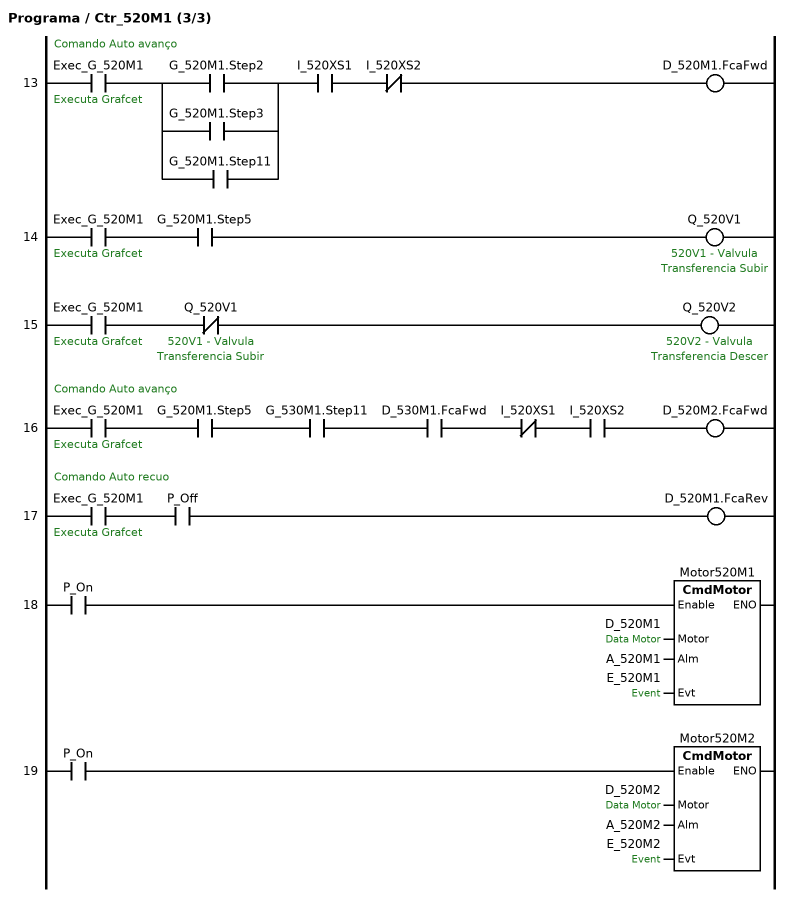
(* [picture p120: Programa / Ctr_520M1, rungs 13-19] *)
(* Rung 13: Comando Auto avanço *)
D_520M1.FcaFwd := Exec_G_520M1 AND (G_520M1.Step2 OR G_520M1.Step3 OR G_520M1.Step11) AND I_520XS1 AND NOT I_520XS2;
(* Rung 14 *)
Q_520V1 := Exec_G_520M1 AND G_520M1.Step5;
(* Rung 15 *)
Q_520V2 := Exec_G_520M1 AND NOT Q_520V1;
(* Rung 16: Comando Auto avanço *)
D_520M2.FcaFwd := Exec_G_520M1 AND G_520M1.Step5 AND G_530M1.Step11 AND D_530M1.FcaFwd AND NOT I_520XS1 AND I_520XS2;
(* Rung 17: Comando Auto recuo *)
D_520M1.FcaRev := Exec_G_520M1 AND P_Off;
(* Rung 18 *)
Motor520M1(Enable := P_On, Motor := D_520M1, Alm := A_520M1, Evt := E_520M1);
(* Rung 19 *)
Motor520M2(Enable := P_On, Motor := D_520M2, Alm := A_520M2, Evt := E_520M2);

(* Section Ctr_530M1: ladder, written here as Structured Text *)

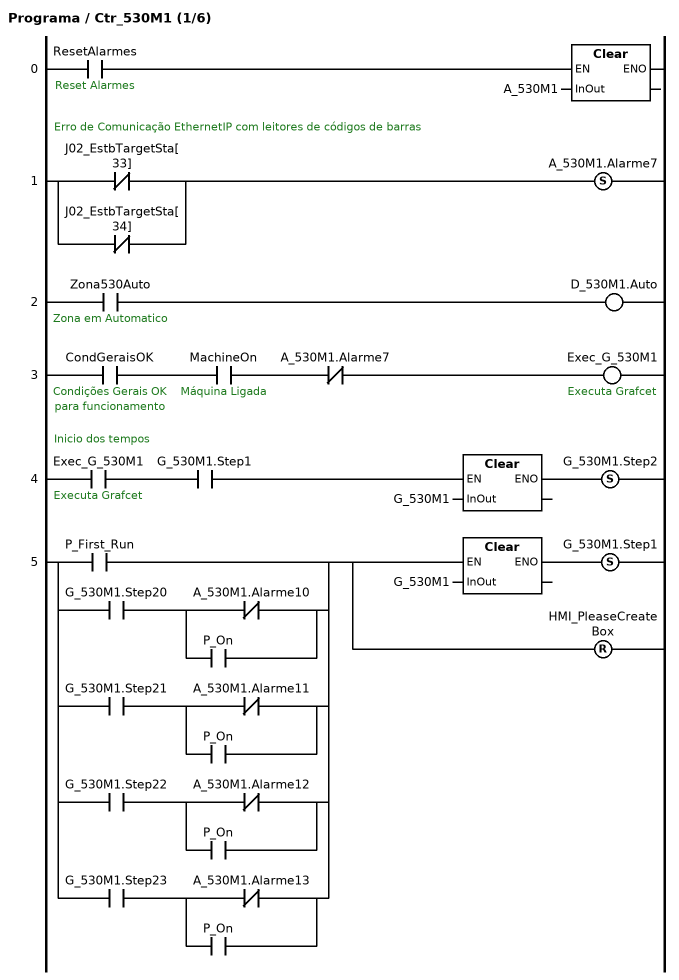
(* Rung 0 *)
IF ResetAlarmes THEN Clear(InOut := A_530M1); END_IF;
(* Rung 1: Erro de Comunicação EthernetIP com leitores de códigos de barras *)
IF NOT J02_EstbTargetSta[33] OR NOT J02_EstbTargetSta[34] THEN A_530M1.Alarme7 := TRUE; END_IF;
(* Rung 2 *)
D_530M1.Auto := Zona530Auto;
(* Rung 3 *)
Exec_G_530M1 := CondGeraisOK AND MachineOn AND NOT A_530M1.Alarme7;
(* Rung 4: Inicio dos tempos *)
_p223 := Exec_G_530M1 AND G_530M1.Step1;
IF _p223 THEN
    Clear(InOut := G_530M1);
    G_530M1.Step2 := TRUE;
END_IF;
(* Rung 5 *)
_p224 := P_First_Run OR (G_530M1.Step20 AND (NOT A_530M1.Alarme10 OR P_On)) OR (G_530M1.Step21 AND (NOT A_530M1.Alarme11 OR P_On)) OR (G_530M1.Step22 AND (NOT A_530M1.Alarme12 OR P_On)) OR (G_530M1.Step23 AND (NOT A_530M1.Alarme13 OR P_On));
IF _p224 THEN
    Clear(InOut := G_530M1);
    G_530M1.Step1 := TRUE;
    HMI_PleaseCreateBox := FALSE;
END_IF;

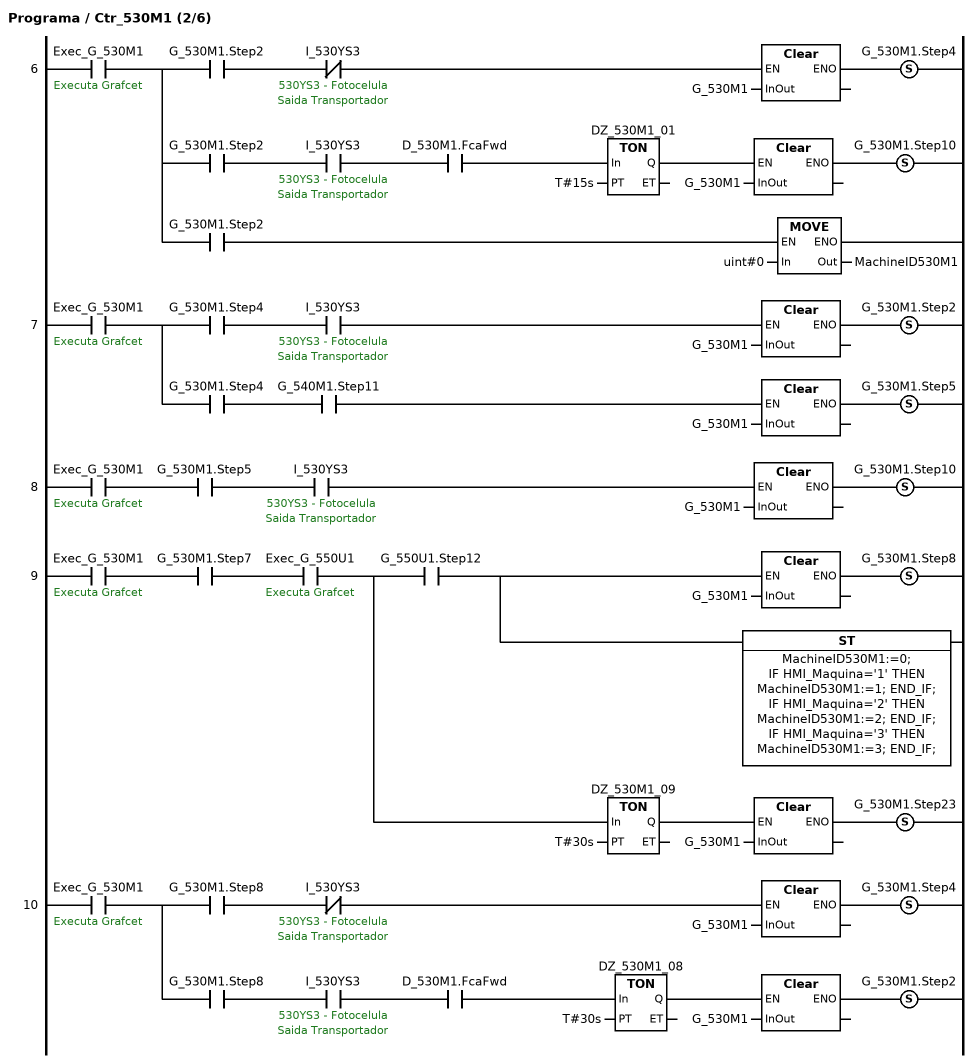
(* Rung 6 *)
_p225 := Exec_G_530M1 AND G_530M1.Step2 AND NOT I_530YS3;
IF _p225 THEN
    Clear(InOut := G_530M1);
    G_530M1.Step4 := TRUE;
END_IF;
DZ_530M1_01(In := Exec_G_530M1 AND G_530M1.Step2 AND I_530YS3 AND D_530M1.FcaFwd, PT := T#15s);
IF DZ_530M1_01.Q THEN
    Clear(InOut := G_530M1);
    G_530M1.Step10 := TRUE;
END_IF;
IF Exec_G_530M1 AND G_530M1.Step2 THEN MachineID530M1 := uint#0; END_IF;
(* Rung 7 *)
_p226 := Exec_G_530M1 AND G_530M1.Step4 AND I_530YS3;
IF _p226 THEN
    Clear(InOut := G_530M1);
    G_530M1.Step2 := TRUE;
END_IF;
_p227 := Exec_G_530M1 AND G_530M1.Step4 AND G_540M1.Step11;
IF _p227 THEN
    Clear(InOut := G_530M1);
    G_530M1.Step5 := TRUE;
END_IF;
(* Rung 8 *)
_p228 := Exec_G_530M1 AND G_530M1.Step5 AND I_530YS3;
IF _p228 THEN
    Clear(InOut := G_530M1);
    G_530M1.Step10 := TRUE;
END_IF;
(* Rung 9 *)
_p229 := Exec_G_530M1 AND G_530M1.Step7 AND Exec_G_550U1 AND G_550U1.Step12;
_p230 := Exec_G_530M1 AND G_530M1.Step7 AND Exec_G_550U1;
IF _p229 THEN
    Clear(InOut := G_530M1);
    G_530M1.Step8 := TRUE;
END_IF;
IF _p229 THEN
    MachineID530M1:=0;
    IF HMI_Maquina='1' THEN MachineID530M1:=1; END_IF;
    IF HMI_Maquina='2' THEN MachineID530M1:=2; END_IF;
    IF HMI_Maquina='3' THEN MachineID530M1:=3; END_IF;
END_IF;
DZ_530M1_09(In := _p230, PT := T#30s);
IF DZ_530M1_09.Q THEN
    Clear(InOut := G_530M1);
    G_530M1.Step23 := TRUE;
END_IF;
(* Rung 10 *)
_p231 := Exec_G_530M1 AND G_530M1.Step8 AND NOT I_530YS3;
IF _p231 THEN
    Clear(InOut := G_530M1);
    G_530M1.Step4 := TRUE;
END_IF;
DZ_530M1_08(In := Exec_G_530M1 AND G_530M1.Step8 AND I_530YS3 AND D_530M1.FcaFwd, PT := T#30s);
IF DZ_530M1_08.Q THEN
    Clear(InOut := G_530M1);
    G_530M1.Step2 := TRUE;
END_IF;

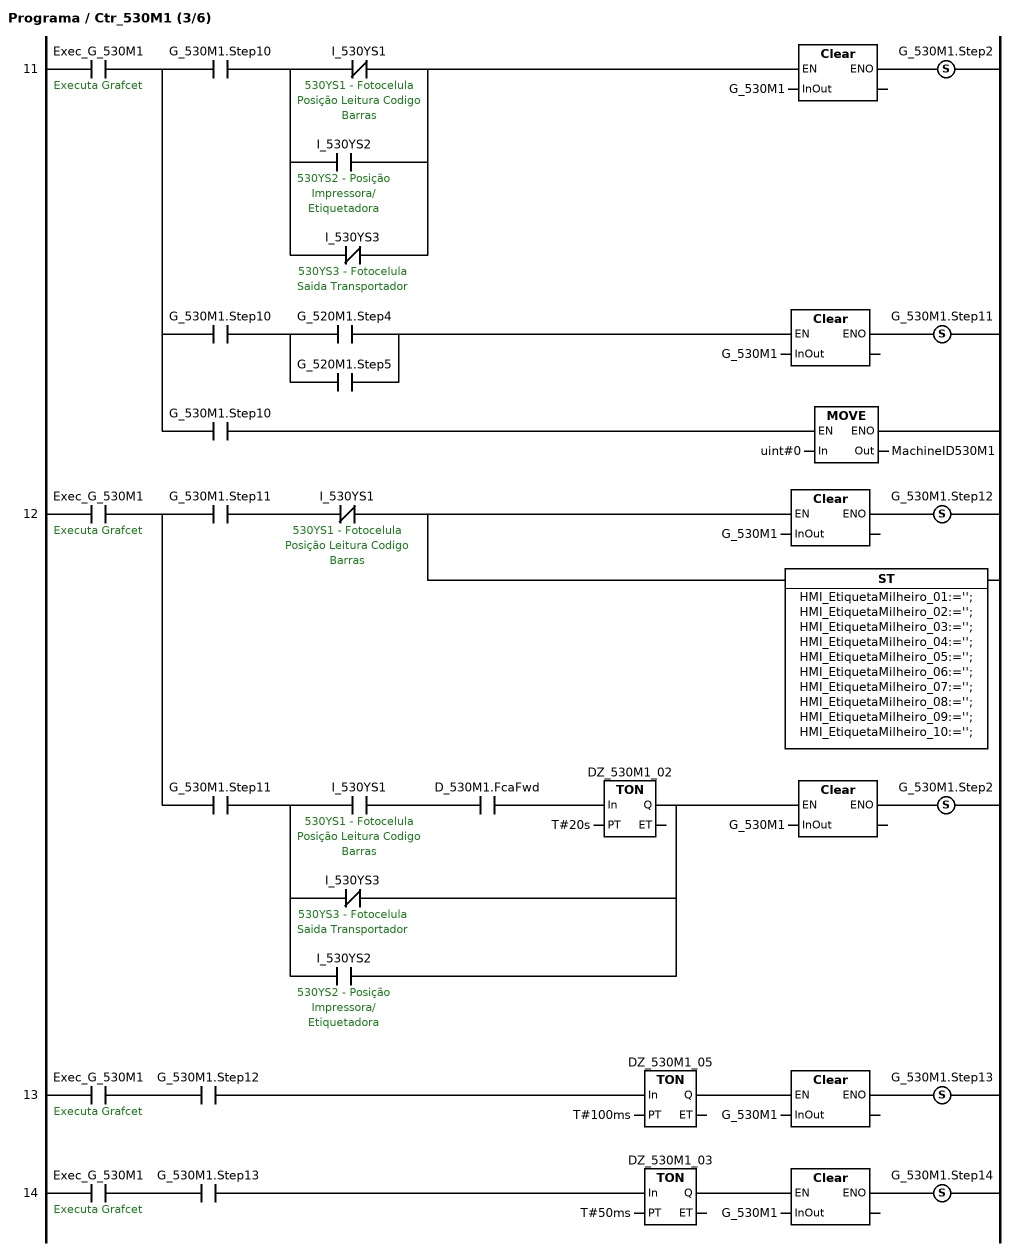
(* Rung 11 *)
_p232 := Exec_G_530M1 AND G_530M1.Step10 AND (NOT I_530YS1 OR I_530YS2 OR NOT I_530YS3);
IF _p232 THEN
    Clear(InOut := G_530M1);
    G_530M1.Step2 := TRUE;
END_IF;
_p233 := Exec_G_530M1 AND G_530M1.Step10 AND (G_520M1.Step4 OR G_520M1.Step5);
IF _p233 THEN
    Clear(InOut := G_530M1);
    G_530M1.Step11 := TRUE;
END_IF;
IF Exec_G_530M1 AND G_530M1.Step10 THEN MachineID530M1 := uint#0; END_IF;
(* Rung 12 *)
_p234 := Exec_G_530M1 AND G_530M1.Step11 AND NOT I_530YS1;
IF _p234 THEN
    Clear(InOut := G_530M1);
    G_530M1.Step12 := TRUE;
END_IF;
IF _p234 THEN
    HMI_EtiquetaMilheiro_01:='';
    HMI_EtiquetaMilheiro_02:='';
    HMI_EtiquetaMilheiro_03:='';
    HMI_EtiquetaMilheiro_04:='';
    HMI_EtiquetaMilheiro_05:='';
    HMI_EtiquetaMilheiro_06:='';
    HMI_EtiquetaMilheiro_07:='';
    HMI_EtiquetaMilheiro_08:='';
    HMI_EtiquetaMilheiro_09:='';
    HMI_EtiquetaMilheiro_10:='';
END_IF;
DZ_530M1_02(In := Exec_G_530M1 AND G_530M1.Step11 AND I_530YS1 AND D_530M1.FcaFwd, PT := T#20s);
_p235 := DZ_530M1_02.Q OR (Exec_G_530M1 AND G_530M1.Step11 AND (NOT I_530YS3 OR I_530YS2));
IF _p235 THEN
    Clear(InOut := G_530M1);
    G_530M1.Step2 := TRUE;
END_IF;
(* Rung 13 *)
DZ_530M1_05(In := Exec_G_530M1 AND G_530M1.Step12, PT := T#100ms);
IF DZ_530M1_05.Q THEN
    Clear(InOut := G_530M1);
    G_530M1.Step13 := TRUE;
END_IF;
(* Rung 14 *)
DZ_530M1_03(In := Exec_G_530M1 AND G_530M1.Step13, PT := T#50ms);
IF DZ_530M1_03.Q THEN
    Clear(InOut := G_530M1);
    G_530M1.Step14 := TRUE;
END_IF;

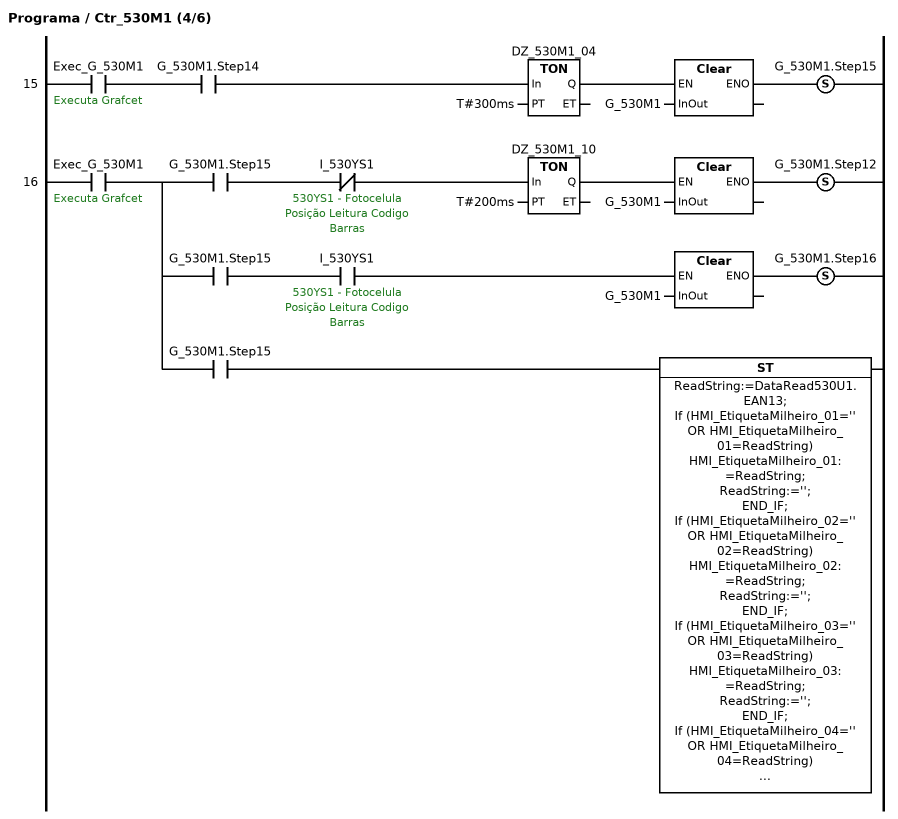
(* Rung 15 *)
DZ_530M1_04(In := Exec_G_530M1 AND G_530M1.Step14, PT := T#300ms);
IF DZ_530M1_04.Q THEN
    Clear(InOut := G_530M1);
    G_530M1.Step15 := TRUE;
END_IF;
(* Rung 16 *)
DZ_530M1_10(In := Exec_G_530M1 AND G_530M1.Step15 AND NOT I_530YS1, PT := T#200ms);
IF DZ_530M1_10.Q THEN
    Clear(InOut := G_530M1);
    G_530M1.Step12 := TRUE;
END_IF;
_p236 := Exec_G_530M1 AND G_530M1.Step15 AND I_530YS1;
IF _p236 THEN
    Clear(InOut := G_530M1);
    G_530M1.Step16 := TRUE;
END_IF;
IF Exec_G_530M1 AND G_530M1.Step15 THEN
    ReadString:=DataRead530U1.EAN13;
    If (HMI_EtiquetaMilheiro_01='' OR HMI_EtiquetaMilheiro_01=ReadString) AND ReadString<>'' THEN
    	HMI_EtiquetaMilheiro_01:=ReadString;
    	ReadString:='';
    END_IF;
    If (HMI_EtiquetaMilheiro_02='' OR HMI_EtiquetaMilheiro_02=ReadString) AND ReadString<>'' THEN
    	HMI_EtiquetaMilheiro_02:=ReadString;
    	ReadString:='';
    END_IF;
    If (HMI_EtiquetaMilheiro_03='' OR HMI_EtiquetaMilheiro_03=ReadString) AND ReadString<>'' THEN
    	HMI_EtiquetaMilheiro_03:=ReadString;
    	ReadString:='';
    END_IF;
    If (HMI_EtiquetaMilheiro_04='' OR HMI_EtiquetaMilheiro_04=ReadString) AND ReadString<>'' THEN
    	HMI_EtiquetaMilheiro_04:=ReadString;
    	ReadString:='';
    END_IF;
    If (HMI_EtiquetaMilheiro_05='' OR HMI_EtiquetaMilheiro_05=ReadString) AND ReadString<>'' THEN
    	HMI_EtiquetaMilheiro_05:=ReadString;
    	ReadString:='';
    END_IF;
    If (HMI_EtiquetaMilheiro_06='' OR HMI_EtiquetaMilheiro_06=ReadString) AND ReadString<>'' THEN
    	HMI_EtiquetaMilheiro_06:=ReadString;
    	ReadString:='';
    END_IF;
    If (HMI_EtiquetaMilheiro_07='' OR HMI_EtiquetaMilheiro_07=ReadString) AND ReadString<>'' THEN
    	HMI_EtiquetaMilheiro_07:=ReadString;
    	ReadString:='';
    END_IF;
    If (HMI_EtiquetaMilheiro_08='' OR HMI_EtiquetaMilheiro_08=ReadString) AND ReadString<>'' THEN
    	HMI_EtiquetaMilheiro_08:=ReadString;
    	ReadString:='';
    END_IF;
    If (HMI_EtiquetaMilheiro_09='' OR HMI_EtiquetaMilheiro_09=ReadString) AND ReadString<>'' THEN
    	HMI_EtiquetaMilheiro_09:=ReadString;
    	ReadString:='';
    END_IF;
    If (HMI_EtiquetaMilheiro_10='' OR HMI_EtiquetaMilheiro_10=ReadString) AND ReadString<>'' THEN
    	HMI_EtiquetaMilheiro_10:=ReadString;
    	ReadString:='';
    END_IF;
    
    ReadString:=DataRead530U2.EAN13;
    If (HMI_EtiquetaMilheiro_01='' OR HMI_EtiquetaMilheiro_01=ReadString) AND ReadString<>'' THEN
    	HMI_EtiquetaMilheiro_01:=ReadString;
    	ReadString:='';
    END_IF;
    If (HMI_EtiquetaMilheiro_02='' OR HMI_EtiquetaMilheiro_02=ReadString) AND ReadString<>'' THEN
    	HMI_EtiquetaMilheiro_02:=ReadString;
    	ReadString:='';
    END_IF;
    If (HMI_EtiquetaMilheiro_03='' OR HMI_EtiquetaMilheiro_03=ReadString) AND ReadString<>'' THEN
    	HMI_EtiquetaMilheiro_03:=ReadString;
    	ReadString:='';
    END_IF;
    If (HMI_EtiquetaMilheiro_04='' OR HMI_EtiquetaMilheiro_04=ReadString) AND ReadString<>'' THEN
    	HMI_EtiquetaMilheiro_04:=ReadString;
    	ReadString:='';
    END_IF;
    If (HMI_EtiquetaMilheiro_05='' OR HMI_EtiquetaMilheiro_05=ReadString) AND ReadString<>'' THEN
    	HMI_EtiquetaMilheiro_05:=ReadString;
    	ReadString:='';
    END_IF;
    If (HMI_EtiquetaMilheiro_06='' OR HMI_EtiquetaMilheiro_06=ReadString) AND ReadString<>'' THEN
    	HMI_EtiquetaMilheiro_06:=ReadString;
    	ReadString:='';
    END_IF;
    If (HMI_EtiquetaMilheiro_07='' OR HMI_EtiquetaMilheiro_07=ReadString) AND ReadString<>'' THEN
    	HMI_EtiquetaMilheiro_07:=ReadString;
    	ReadString:='';
    END_IF;
    If (HMI_EtiquetaMilheiro_08='' OR HMI_EtiquetaMilheiro_08=ReadString) AND ReadString<>'' THEN
    	HMI_EtiquetaMilheiro_08:=ReadString;
    	ReadString:='';
    END_IF;
    If (HMI_EtiquetaMilheiro_09='' OR HMI_EtiquetaMilheiro_09=ReadString) AND ReadString<>'' THEN
    	HMI_EtiquetaMilheiro_09:=ReadString;
    	ReadString:='';
    END_IF;
    If (HMI_EtiquetaMilheiro_10='' OR HMI_EtiquetaMilheiro_10=ReadString) AND ReadString<>'' THEN
    	HMI_EtiquetaMilheiro_10:=ReadString;
    	ReadString:='';
    END_IF;
END_IF;

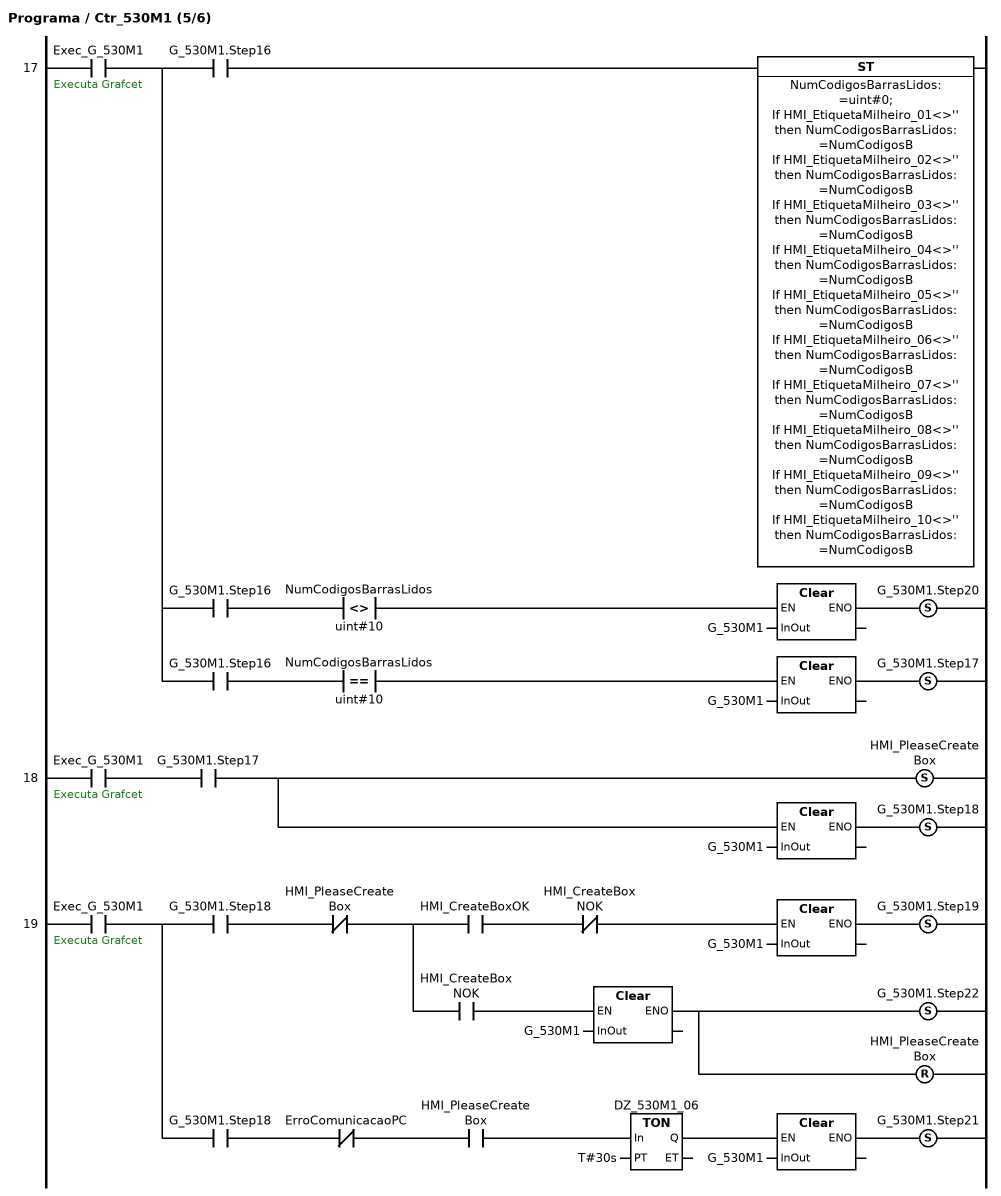
(* Rung 17 *)
IF Exec_G_530M1 AND G_530M1.Step16 THEN
    NumCodigosBarrasLidos:=uint#0;
    If HMI_EtiquetaMilheiro_01<>'' then NumCodigosBarrasLidos:=NumCodigosBarrasLidos+1; END_IF;
    If HMI_EtiquetaMilheiro_02<>'' then NumCodigosBarrasLidos:=NumCodigosBarrasLidos+1; END_IF;
    If HMI_EtiquetaMilheiro_03<>'' then NumCodigosBarrasLidos:=NumCodigosBarrasLidos+1; END_IF;
    If HMI_EtiquetaMilheiro_04<>'' then NumCodigosBarrasLidos:=NumCodigosBarrasLidos+1; END_IF;
    If HMI_EtiquetaMilheiro_05<>'' then NumCodigosBarrasLidos:=NumCodigosBarrasLidos+1; END_IF;
    If HMI_EtiquetaMilheiro_06<>'' then NumCodigosBarrasLidos:=NumCodigosBarrasLidos+1; END_IF;
    If HMI_EtiquetaMilheiro_07<>'' then NumCodigosBarrasLidos:=NumCodigosBarrasLidos+1; END_IF;
    If HMI_EtiquetaMilheiro_08<>'' then NumCodigosBarrasLidos:=NumCodigosBarrasLidos+1; END_IF;
    If HMI_EtiquetaMilheiro_09<>'' then NumCodigosBarrasLidos:=NumCodigosBarrasLidos+1; END_IF;
    If HMI_EtiquetaMilheiro_10<>'' then NumCodigosBarrasLidos:=NumCodigosBarrasLidos+1; END_IF;
END_IF;
_p237 := Exec_G_530M1 AND G_530M1.Step16 AND (NumCodigosBarrasLidos <> uint#10);
IF _p237 THEN
    Clear(InOut := G_530M1);
    G_530M1.Step20 := TRUE;
END_IF;
_p238 := Exec_G_530M1 AND G_530M1.Step16 AND (NumCodigosBarrasLidos = uint#10);
IF _p238 THEN
    Clear(InOut := G_530M1);
    G_530M1.Step17 := TRUE;
END_IF;
(* Rung 18 *)
IF Exec_G_530M1 AND G_530M1.Step17 THEN HMI_PleaseCreateBox := TRUE; END_IF;
_p239 := Exec_G_530M1 AND G_530M1.Step17;
IF _p239 THEN
    Clear(InOut := G_530M1);
    G_530M1.Step18 := TRUE;
END_IF;
(* Rung 19 *)
_p240 := Exec_G_530M1 AND G_530M1.Step18 AND NOT HMI_PleaseCreateBox;
IF _p240 AND HMI_CreateBoxOK AND NOT HMI_CreateBoxNOK THEN
    Clear(InOut := G_530M1);
    G_530M1.Step19 := TRUE;
END_IF;
IF _p240 AND HMI_CreateBoxNOK THEN
    Clear(InOut := G_530M1);
    G_530M1.Step22 := TRUE;
    HMI_PleaseCreateBox := FALSE;
END_IF;
DZ_530M1_06(In := Exec_G_530M1 AND G_530M1.Step18 AND NOT ErroComunicacaoPC AND HMI_PleaseCreateBox, PT := T#30s);
IF DZ_530M1_06.Q THEN
    Clear(InOut := G_530M1);
    G_530M1.Step21 := TRUE;
END_IF;

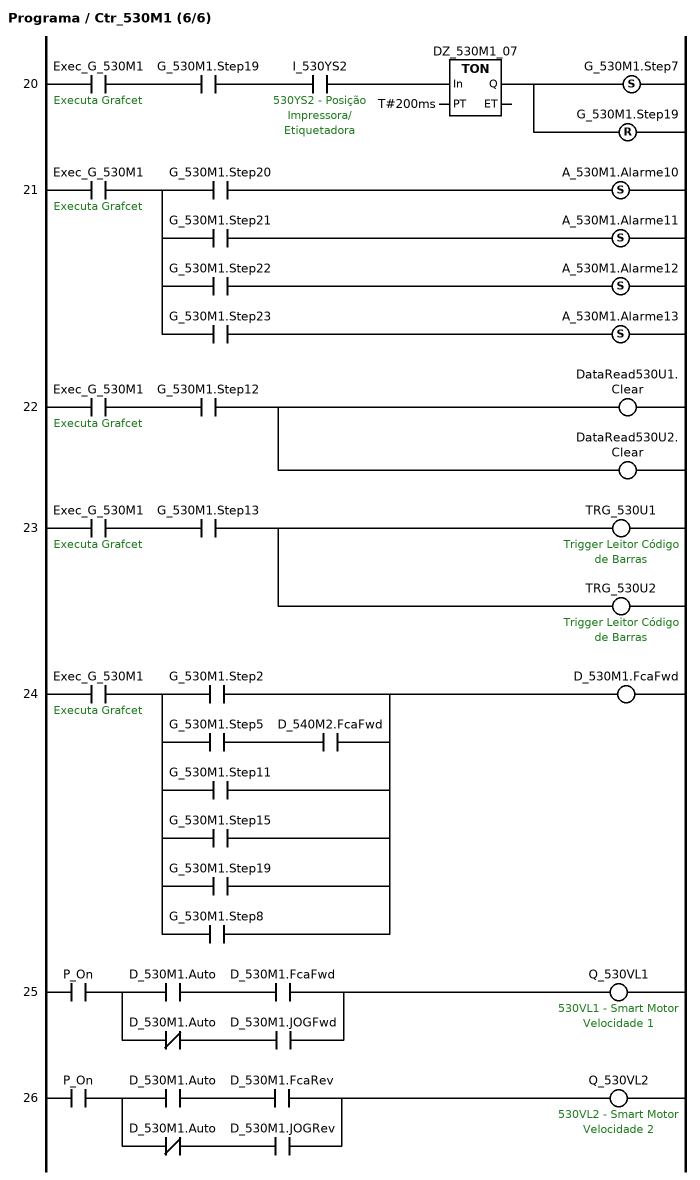
(* Rung 20 *)
DZ_530M1_07(In := Exec_G_530M1 AND G_530M1.Step19 AND I_530YS2, PT := T#200ms);
IF DZ_530M1_07.Q THEN
    G_530M1.Step7 := TRUE;
    G_530M1.Step19 := FALSE;
END_IF;
(* Rung 21 *)
IF Exec_G_530M1 AND G_530M1.Step20 THEN A_530M1.Alarme10 := TRUE; END_IF;
IF Exec_G_530M1 AND G_530M1.Step21 THEN A_530M1.Alarme11 := TRUE; END_IF;
IF Exec_G_530M1 AND G_530M1.Step22 THEN A_530M1.Alarme12 := TRUE; END_IF;
IF Exec_G_530M1 AND G_530M1.Step23 THEN A_530M1.Alarme13 := TRUE; END_IF;
(* Rung 22 *)
DataRead530U1.Clear := Exec_G_530M1 AND G_530M1.Step12;
DataRead530U2.Clear := Exec_G_530M1 AND G_530M1.Step12;
(* Rung 23 *)
TRG_530U1 := Exec_G_530M1 AND G_530M1.Step13;
TRG_530U2 := Exec_G_530M1 AND G_530M1.Step13;
(* Rung 24 *)
D_530M1.FcaFwd := Exec_G_530M1 AND (G_530M1.Step2 OR (G_530M1.Step5 AND D_540M2.FcaFwd) OR G_530M1.Step11 OR G_530M1.Step15 OR G_530M1.Step19 OR G_530M1.Step8);
(* Rung 25 *)
Q_530VL1 := P_On AND ((D_530M1.Auto AND D_530M1.FcaFwd) OR (NOT D_530M1.Auto AND D_530M1.JOGFwd));
(* Rung 26 *)
Q_530VL2 := P_On AND ((D_530M1.Auto AND D_530M1.FcaRev) OR (NOT D_530M1.Auto AND D_530M1.JOGRev));

(* Section Data530U1_Scanner: ladder, written here as Structured Text *)

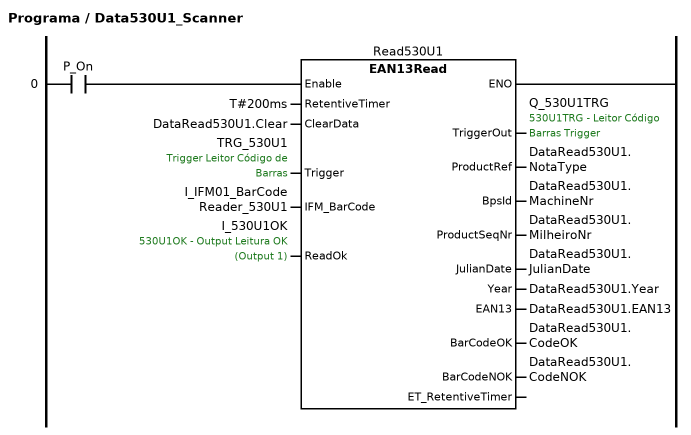
(* Rung 0 *)
Read530U1(Enable := P_On, RetentiveTimer := T#200ms, ClearData := DataRead530U1.Clear, Trigger := TRG_530U1, IFM_BarCode := I_IFM01_BarCodeReader_530U1, ReadOk := I_530U1OK, TriggerOut => Q_530U1TRG, ProductRef => DataRead530U1.NotaType, BpsId => DataRead530U1.MachineNr, ProductSeqNr => DataRead530U1.MilheiroNr, JulianDate => DataRead530U1.JulianDate, Year => DataRead530U1.Year, EAN13 => DataRead530U1.EAN13, BarCodeOK => DataRead530U1.CodeOK, BarCodeNOK => DataRead530U1.CodeNOK);

(* Section Data530U2_Scanner: ladder, written here as Structured Text *)

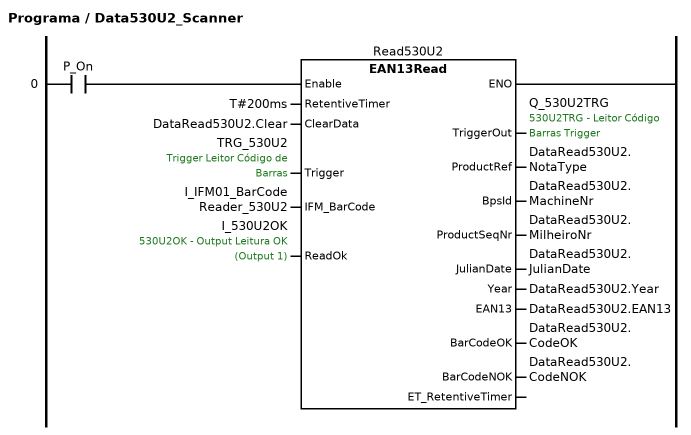
(* Rung 0 *)
Read530U2(Enable := P_On, RetentiveTimer := T#200ms, ClearData := DataRead530U2.Clear, Trigger := TRG_530U2, IFM_BarCode := I_IFM01_BarCodeReader_530U2, ReadOk := I_530U2OK, TriggerOut => Q_530U2TRG, ProductRef => DataRead530U2.NotaType, BpsId => DataRead530U2.MachineNr, ProductSeqNr => DataRead530U2.MilheiroNr, JulianDate => DataRead530U2.JulianDate, Year => DataRead530U2.Year, EAN13 => DataRead530U2.EAN13, BarCodeOK => DataRead530U2.CodeOK, BarCodeNOK => DataRead530U2.CodeNOK);

(* Section Ctr_540M1: ladder, written here as Structured Text *)

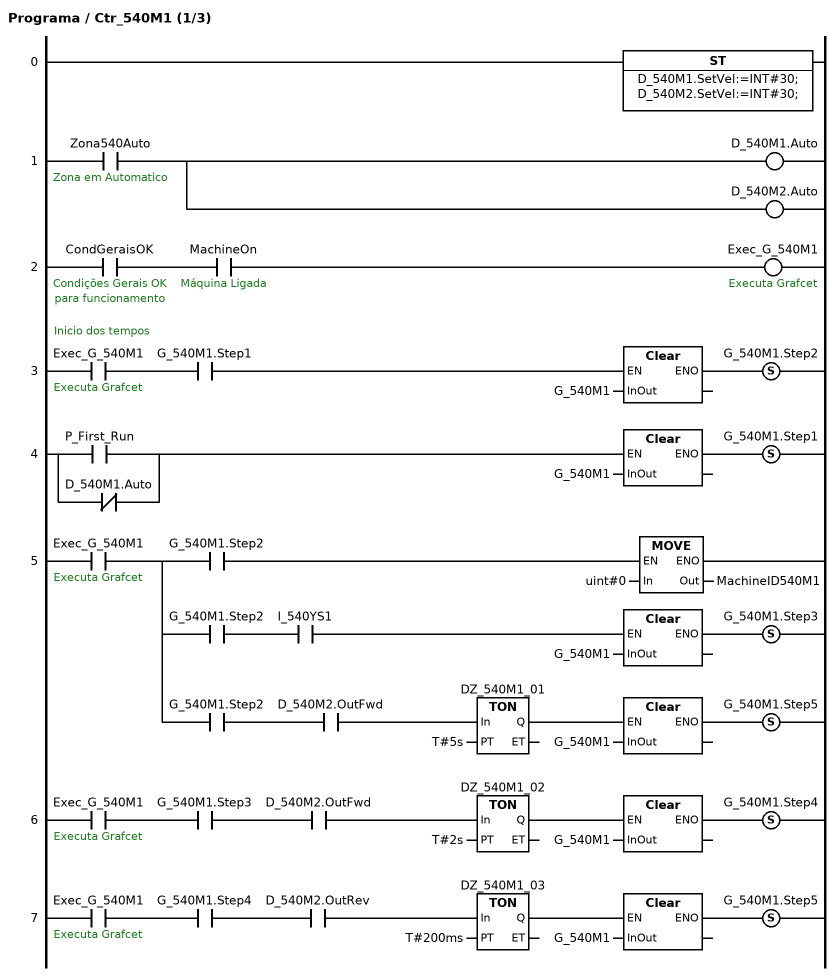
(* Rung 0 *)
D_540M1.SetVel:=INT#30;
D_540M2.SetVel:=INT#30;
(* Rung 1 *)
D_540M1.Auto := Zona540Auto;
D_540M2.Auto := Zona540Auto;
(* Rung 2 *)
Exec_G_540M1 := CondGeraisOK AND MachineOn;
(* Rung 3: Inicio dos tempos *)
_p241 := Exec_G_540M1 AND G_540M1.Step1;
IF _p241 THEN
    Clear(InOut := G_540M1);
    G_540M1.Step2 := TRUE;
END_IF;
(* Rung 4 *)
IF P_First_Run OR NOT D_540M1.Auto THEN
    Clear(InOut := G_540M1);
    G_540M1.Step1 := TRUE;
END_IF;
(* Rung 5 *)
IF Exec_G_540M1 AND G_540M1.Step2 THEN MachineID540M1 := uint#0; END_IF;
_p242 := Exec_G_540M1 AND G_540M1.Step2 AND I_540YS1;
IF _p242 THEN
    Clear(InOut := G_540M1);
    G_540M1.Step3 := TRUE;
END_IF;
DZ_540M1_01(In := Exec_G_540M1 AND G_540M1.Step2 AND D_540M2.OutFwd, PT := T#5s);
IF DZ_540M1_01.Q THEN
    Clear(InOut := G_540M1);
    G_540M1.Step5 := TRUE;
END_IF;
(* Rung 6 *)
DZ_540M1_02(In := Exec_G_540M1 AND G_540M1.Step3 AND D_540M2.OutFwd, PT := T#2s);
IF DZ_540M1_02.Q THEN
    Clear(InOut := G_540M1);
    G_540M1.Step4 := TRUE;
END_IF;
(* Rung 7 *)
DZ_540M1_03(In := Exec_G_540M1 AND G_540M1.Step4 AND D_540M2.OutRev, PT := T#200ms);
IF DZ_540M1_03.Q THEN
    Clear(InOut := G_540M1);
    G_540M1.Step5 := TRUE;
END_IF;

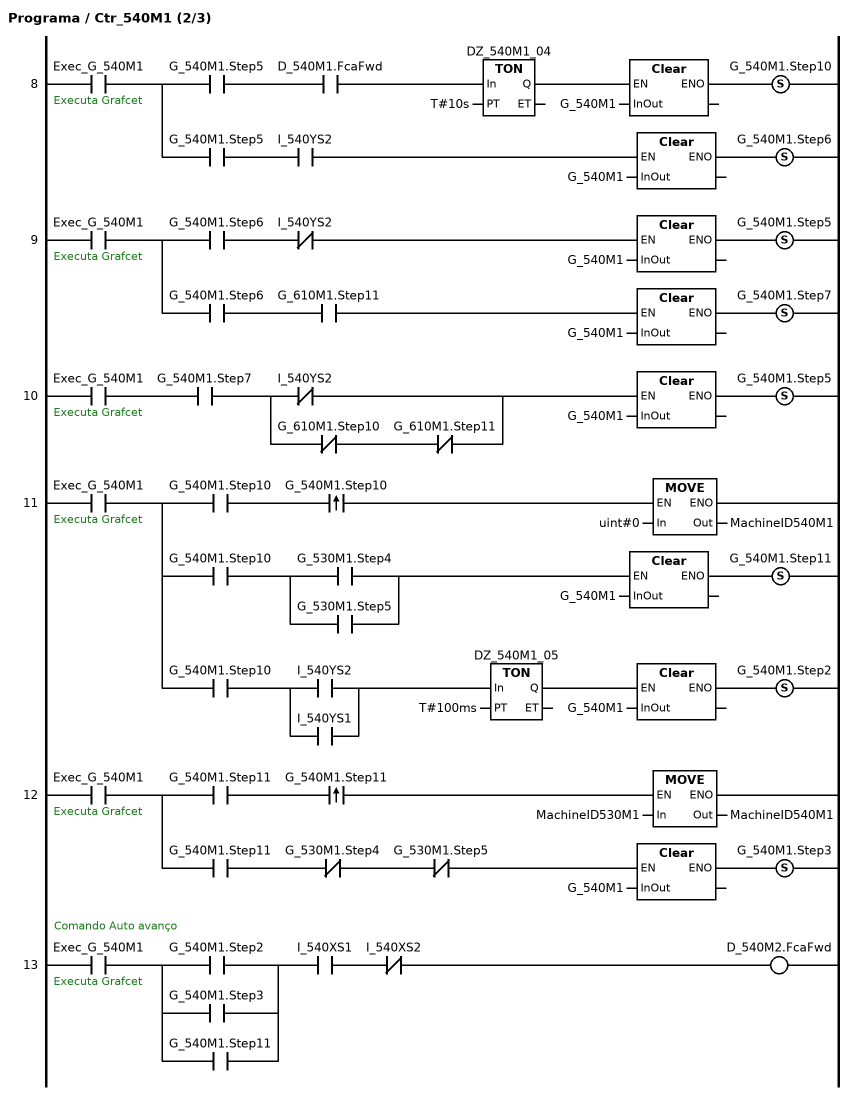
(* Rung 8 *)
DZ_540M1_04(In := Exec_G_540M1 AND G_540M1.Step5 AND D_540M1.FcaFwd, PT := T#10s);
IF DZ_540M1_04.Q THEN
    Clear(InOut := G_540M1);
    G_540M1.Step10 := TRUE;
END_IF;
_p243 := Exec_G_540M1 AND G_540M1.Step5 AND I_540YS2;
IF _p243 THEN
    Clear(InOut := G_540M1);
    G_540M1.Step6 := TRUE;
END_IF;
(* Rung 9 *)
_p244 := Exec_G_540M1 AND G_540M1.Step6 AND NOT I_540YS2;
IF _p244 THEN
    Clear(InOut := G_540M1);
    G_540M1.Step5 := TRUE;
END_IF;
_p245 := Exec_G_540M1 AND G_540M1.Step6 AND G_610M1.Step11;
IF _p245 THEN
    Clear(InOut := G_540M1);
    G_540M1.Step7 := TRUE;
END_IF;
(* Rung 10 *)
_p246 := Exec_G_540M1 AND G_540M1.Step7 AND (NOT I_540YS2 OR (NOT G_610M1.Step10 AND NOT G_610M1.Step11));
IF _p246 THEN
    Clear(InOut := G_540M1);
    G_540M1.Step5 := TRUE;
END_IF;
(* Rung 11 *)
_e247(CLK := G_540M1.Step10);
IF Exec_G_540M1 AND G_540M1.Step10 AND _e247.Q THEN MachineID540M1 := uint#0; END_IF;
_p248 := Exec_G_540M1 AND G_540M1.Step10 AND (G_530M1.Step4 OR G_530M1.Step5);
IF _p248 THEN
    Clear(InOut := G_540M1);
    G_540M1.Step11 := TRUE;
END_IF;
DZ_540M1_05(In := Exec_G_540M1 AND G_540M1.Step10 AND (I_540YS2 OR I_540YS1), PT := T#100ms);
IF DZ_540M1_05.Q THEN
    Clear(InOut := G_540M1);
    G_540M1.Step2 := TRUE;
END_IF;
(* Rung 12 *)
_e249(CLK := G_540M1.Step11);
IF Exec_G_540M1 AND G_540M1.Step11 AND _e249.Q THEN MachineID540M1 := MachineID530M1; END_IF;
_p250 := Exec_G_540M1 AND G_540M1.Step11 AND NOT G_530M1.Step4 AND NOT G_530M1.Step5;
IF _p250 THEN
    Clear(InOut := G_540M1);
    G_540M1.Step3 := TRUE;
END_IF;
(* Rung 13: Comando Auto avanço *)
D_540M2.FcaFwd := Exec_G_540M1 AND (G_540M1.Step2 OR G_540M1.Step3 OR G_540M1.Step11) AND I_540XS1 AND NOT I_540XS2;

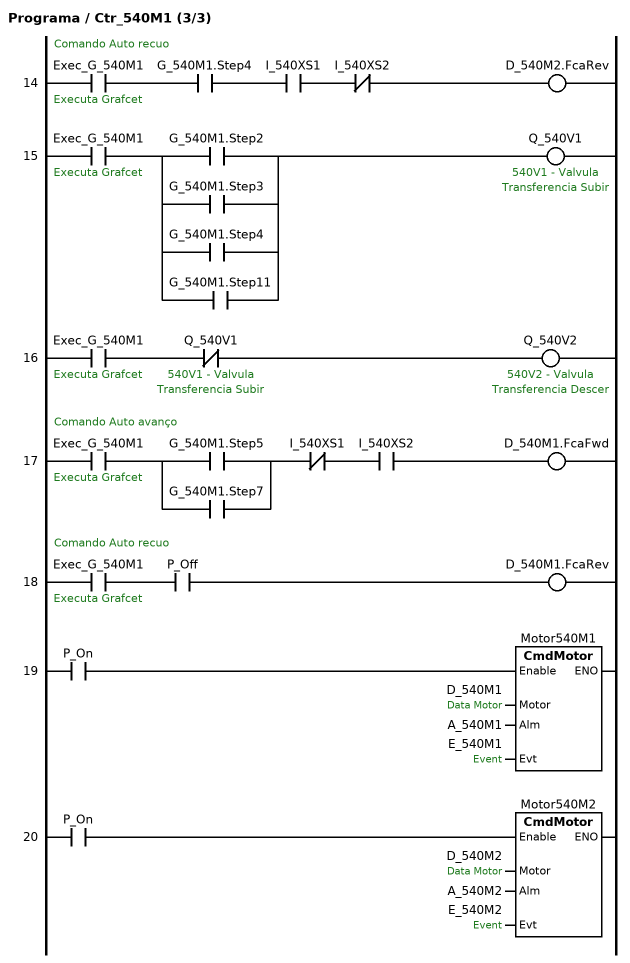
(* Rung 14: Comando Auto recuo *)
D_540M2.FcaRev := Exec_G_540M1 AND G_540M1.Step4 AND I_540XS1 AND NOT I_540XS2;
(* Rung 15 *)
Q_540V1 := Exec_G_540M1 AND (G_540M1.Step2 OR G_540M1.Step3 OR G_540M1.Step4 OR G_540M1.Step11);
(* Rung 16 *)
Q_540V2 := Exec_G_540M1 AND NOT Q_540V1;
(* Rung 17: Comando Auto avanço *)
D_540M1.FcaFwd := Exec_G_540M1 AND (G_540M1.Step5 OR G_540M1.Step7) AND NOT I_540XS1 AND I_540XS2;
(* Rung 18: Comando Auto recuo *)
D_540M1.FcaRev := Exec_G_540M1 AND P_Off;
(* Rung 19 *)
Motor540M1(Enable := P_On, Motor := D_540M1, Alm := A_540M1, Evt := E_540M1);
(* Rung 20 *)
Motor540M2(Enable := P_On, Motor := D_540M2, Alm := A_540M2, Evt := E_540M2);

(* Section Ctr_550U1_Impressora: ladder, written here as Structured Text *)

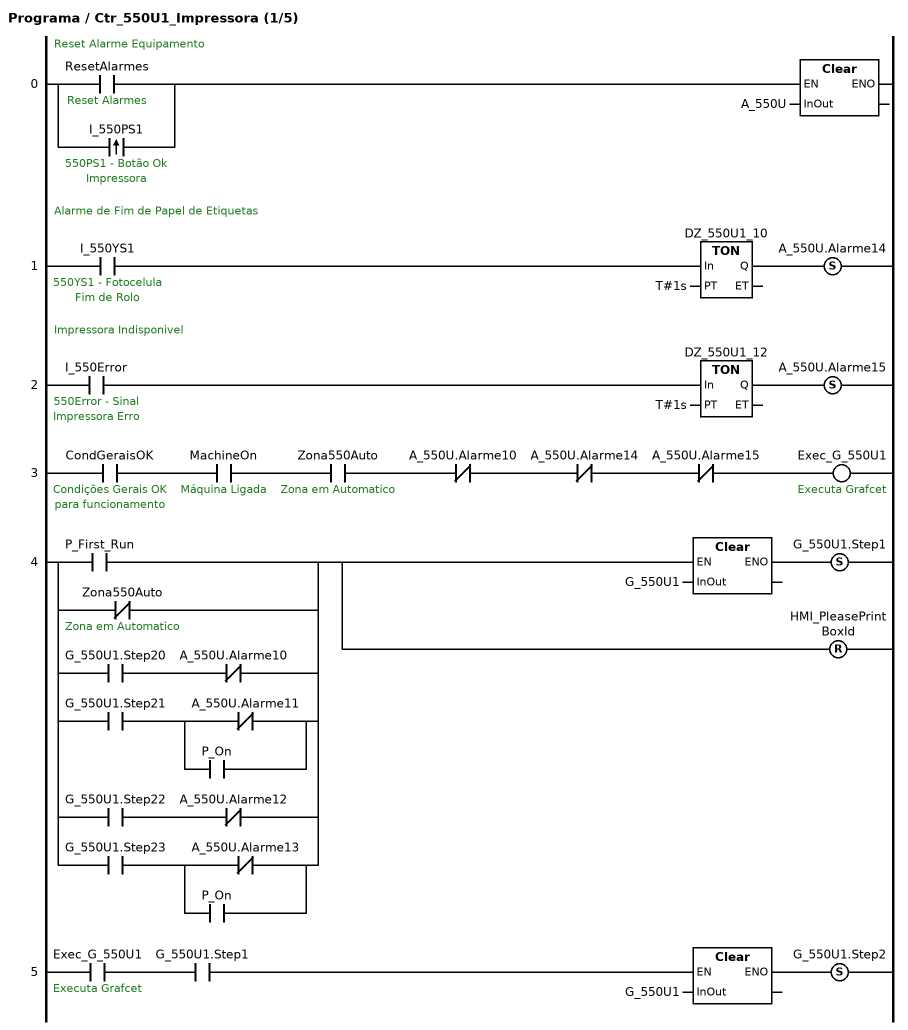
(* Rung 0: Reset Alarme Equipamento *)
_e251(CLK := I_550PS1);
IF ResetAlarmes OR _e251.Q THEN Clear(InOut := A_550U); END_IF;
(* Rung 1: Alarme de Fim de Papel de Etiquetas *)
DZ_550U1_10(In := I_550YS1, PT := T#1s);
IF DZ_550U1_10.Q THEN A_550U.Alarme14 := TRUE; END_IF;
(* Rung 2: Impressora Indisponivel *)
DZ_550U1_12(In := I_550Error, PT := T#1s);
IF DZ_550U1_12.Q THEN A_550U.Alarme15 := TRUE; END_IF;
(* Rung 3 *)
Exec_G_550U1 := CondGeraisOK AND MachineOn AND Zona550Auto AND NOT A_550U.Alarme10 AND NOT A_550U.Alarme14 AND NOT A_550U.Alarme15;
(* Rung 4 *)
_p252 := P_First_Run OR NOT Zona550Auto OR (G_550U1.Step20 AND NOT A_550U.Alarme10) OR (G_550U1.Step21 AND (NOT A_550U.Alarme11 OR P_On)) OR (G_550U1.Step22 AND NOT A_550U.Alarme12) OR (G_550U1.Step23 AND (NOT A_550U.Alarme13 OR P_On));
IF _p252 THEN
    Clear(InOut := G_550U1);
    G_550U1.Step1 := TRUE;
    HMI_PleasePrintBoxId := FALSE;
END_IF;
(* Rung 5 *)
_p253 := Exec_G_550U1 AND G_550U1.Step1;
IF _p253 THEN
    Clear(InOut := G_550U1);
    G_550U1.Step2 := TRUE;
END_IF;

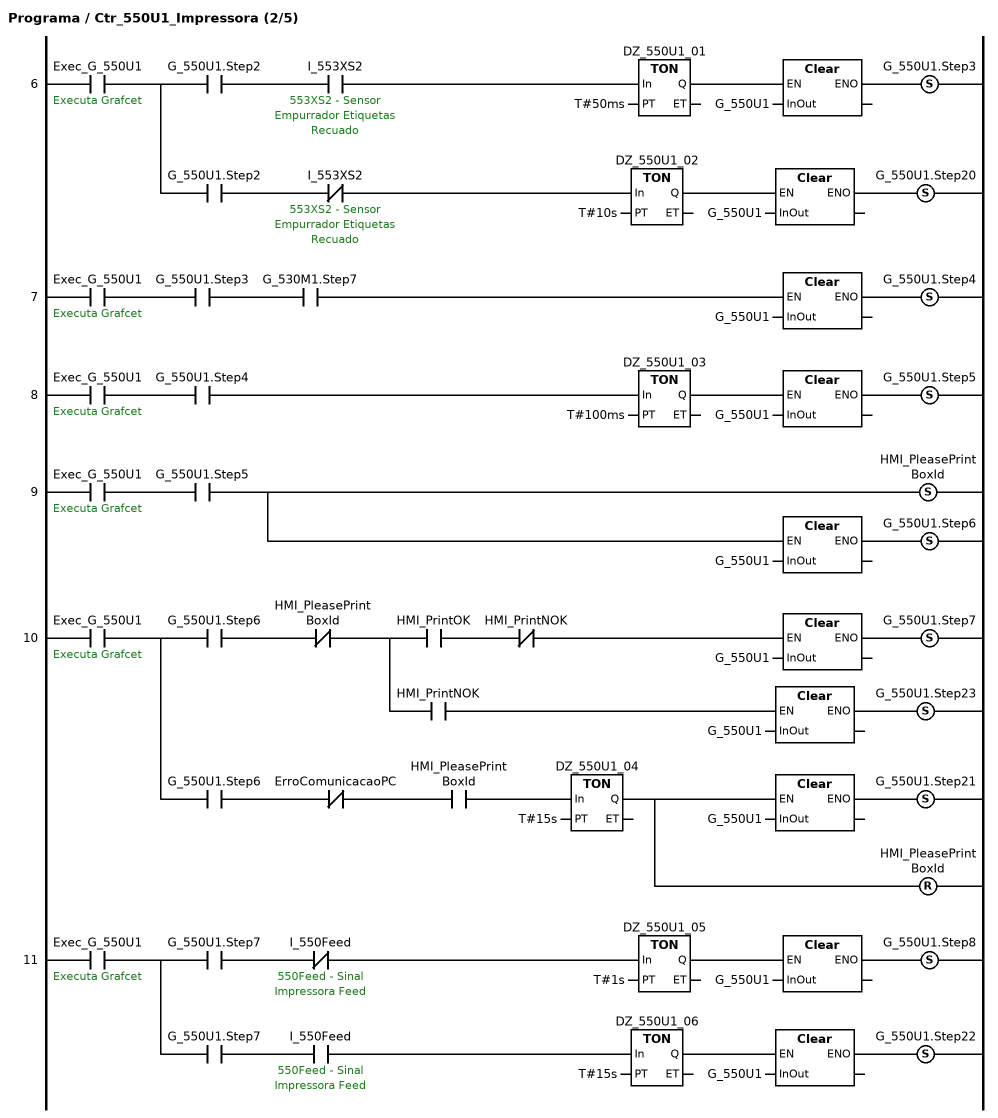
(* Rung 6 *)
DZ_550U1_01(In := Exec_G_550U1 AND G_550U1.Step2 AND I_553XS2, PT := T#50ms);
IF DZ_550U1_01.Q THEN
    Clear(InOut := G_550U1);
    G_550U1.Step3 := TRUE;
END_IF;
DZ_550U1_02(In := Exec_G_550U1 AND G_550U1.Step2 AND NOT I_553XS2, PT := T#10s);
IF DZ_550U1_02.Q THEN
    Clear(InOut := G_550U1);
    G_550U1.Step20 := TRUE;
END_IF;
(* Rung 7 *)
_p254 := Exec_G_550U1 AND G_550U1.Step3 AND G_530M1.Step7;
IF _p254 THEN
    Clear(InOut := G_550U1);
    G_550U1.Step4 := TRUE;
END_IF;
(* Rung 8 *)
DZ_550U1_03(In := Exec_G_550U1 AND G_550U1.Step4, PT := T#100ms);
IF DZ_550U1_03.Q THEN
    Clear(InOut := G_550U1);
    G_550U1.Step5 := TRUE;
END_IF;
(* Rung 9 *)
IF Exec_G_550U1 AND G_550U1.Step5 THEN HMI_PleasePrintBoxId := TRUE; END_IF;
_p255 := Exec_G_550U1 AND G_550U1.Step5;
IF _p255 THEN
    Clear(InOut := G_550U1);
    G_550U1.Step6 := TRUE;
END_IF;
(* Rung 10 *)
_p256 := Exec_G_550U1 AND G_550U1.Step6 AND NOT HMI_PleasePrintBoxId;
IF _p256 AND HMI_PrintOK AND NOT HMI_PrintNOK THEN
    Clear(InOut := G_550U1);
    G_550U1.Step7 := TRUE;
END_IF;
IF _p256 AND HMI_PrintNOK THEN
    Clear(InOut := G_550U1);
    G_550U1.Step23 := TRUE;
END_IF;
DZ_550U1_04(In := Exec_G_550U1 AND G_550U1.Step6 AND NOT ErroComunicacaoPC AND HMI_PleasePrintBoxId, PT := T#15s);
IF DZ_550U1_04.Q THEN
    Clear(InOut := G_550U1);
    G_550U1.Step21 := TRUE;
    HMI_PleasePrintBoxId := FALSE;
END_IF;
(* Rung 11 *)
DZ_550U1_05(In := Exec_G_550U1 AND G_550U1.Step7 AND NOT I_550Feed, PT := T#1s);
IF DZ_550U1_05.Q THEN
    Clear(InOut := G_550U1);
    G_550U1.Step8 := TRUE;
END_IF;
DZ_550U1_06(In := Exec_G_550U1 AND G_550U1.Step7 AND I_550Feed, PT := T#15s);
IF DZ_550U1_06.Q THEN
    Clear(InOut := G_550U1);
    G_550U1.Step22 := TRUE;
END_IF;

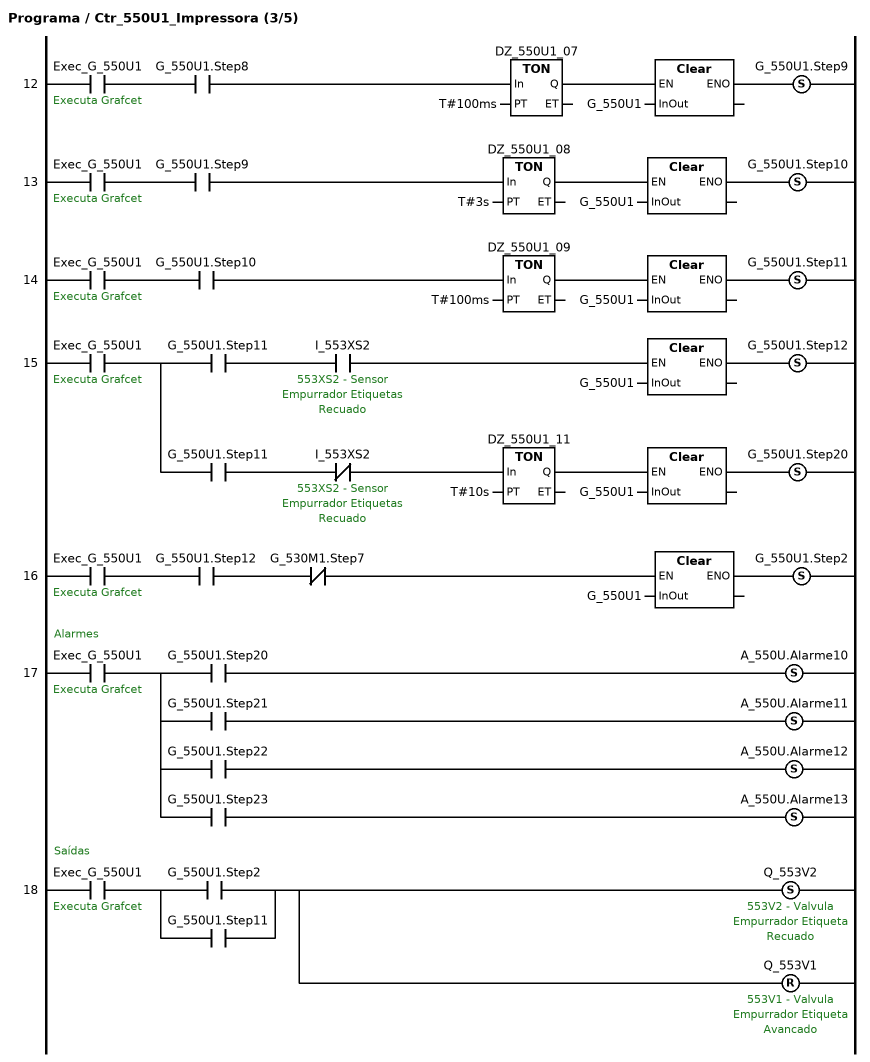
(* Rung 12 *)
DZ_550U1_07(In := Exec_G_550U1 AND G_550U1.Step8, PT := T#100ms);
IF DZ_550U1_07.Q THEN
    Clear(InOut := G_550U1);
    G_550U1.Step9 := TRUE;
END_IF;
(* Rung 13 *)
DZ_550U1_08(In := Exec_G_550U1 AND G_550U1.Step9, PT := T#3s);
IF DZ_550U1_08.Q THEN
    Clear(InOut := G_550U1);
    G_550U1.Step10 := TRUE;
END_IF;
(* Rung 14 *)
DZ_550U1_09(In := Exec_G_550U1 AND G_550U1.Step10, PT := T#100ms);
IF DZ_550U1_09.Q THEN
    Clear(InOut := G_550U1);
    G_550U1.Step11 := TRUE;
END_IF;
(* Rung 15 *)
_p257 := Exec_G_550U1 AND G_550U1.Step11 AND I_553XS2;
IF _p257 THEN
    Clear(InOut := G_550U1);
    G_550U1.Step12 := TRUE;
END_IF;
DZ_550U1_11(In := Exec_G_550U1 AND G_550U1.Step11 AND NOT I_553XS2, PT := T#10s);
IF DZ_550U1_11.Q THEN
    Clear(InOut := G_550U1);
    G_550U1.Step20 := TRUE;
END_IF;
(* Rung 16 *)
_p258 := Exec_G_550U1 AND G_550U1.Step12 AND NOT G_530M1.Step7;
IF _p258 THEN
    Clear(InOut := G_550U1);
    G_550U1.Step2 := TRUE;
END_IF;
(* Rung 17: Alarmes *)
IF Exec_G_550U1 AND G_550U1.Step20 THEN A_550U.Alarme10 := TRUE; END_IF;
IF Exec_G_550U1 AND G_550U1.Step21 THEN A_550U.Alarme11 := TRUE; END_IF;
IF Exec_G_550U1 AND G_550U1.Step22 THEN A_550U.Alarme12 := TRUE; END_IF;
IF Exec_G_550U1 AND G_550U1.Step23 THEN A_550U.Alarme13 := TRUE; END_IF;
(* Rung 18: Saídas *)
_p259 := Exec_G_550U1 AND (G_550U1.Step2 OR G_550U1.Step11);
IF _p259 THEN
    Q_553V2 := TRUE;
    Q_553V1 := FALSE;
END_IF;

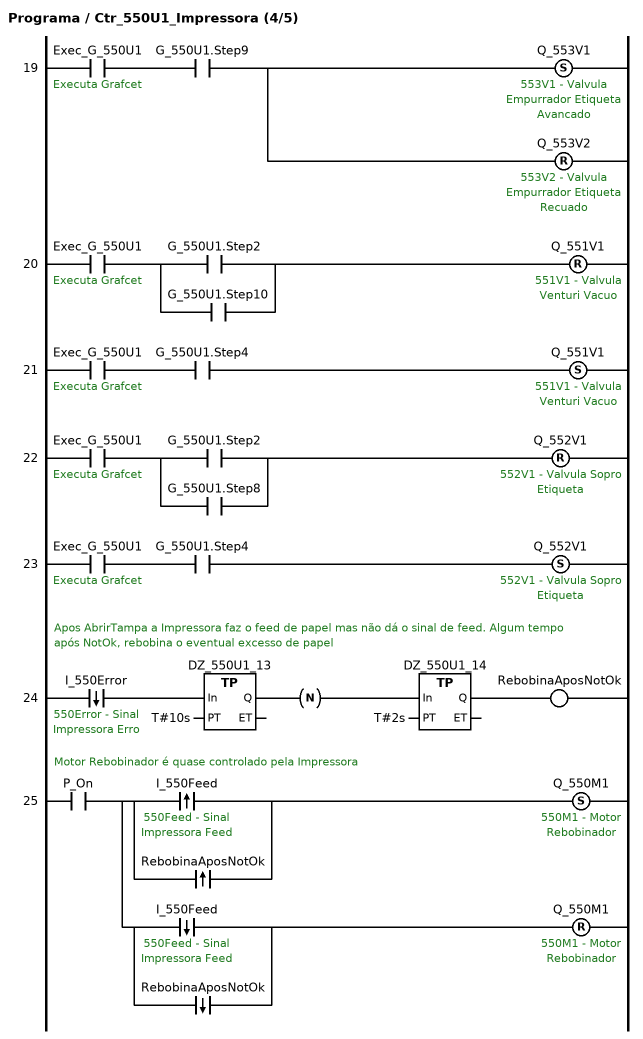
(* Rung 19 *)
IF Exec_G_550U1 AND G_550U1.Step9 THEN
    Q_553V1 := TRUE;
    Q_553V2 := FALSE;
END_IF;
(* Rung 20 *)
IF Exec_G_550U1 AND (G_550U1.Step2 OR G_550U1.Step10) THEN Q_551V1 := FALSE; END_IF;
(* Rung 21 *)
IF Exec_G_550U1 AND G_550U1.Step4 THEN Q_551V1 := TRUE; END_IF;
(* Rung 22 *)
IF Exec_G_550U1 AND (G_550U1.Step2 OR G_550U1.Step8) THEN Q_552V1 := FALSE; END_IF;
(* Rung 23 *)
IF Exec_G_550U1 AND G_550U1.Step4 THEN Q_552V1 := TRUE; END_IF;
(* Rung 24: Apos AbrirTampa a Impressora faz o feed de papel mas não dá o sinal de feed. Algum tempo após NotOk, rebobina o eventual excesso de papel *)
_e260(CLK := I_550Error);
DZ_550U1_13(In := _e260.Q, PT := T#10s);
_e261(CLK := DZ_550U1_13.Q);
DZ_550U1_14(In := _e261.Q, PT := T#2s);
RebobinaAposNotOk := DZ_550U1_14.Q;
(* Rung 25: Motor Rebobinador é quase controlado pela Impressora *)
_e262(CLK := I_550Feed);
_e263(CLK := RebobinaAposNotOk);
IF P_On AND (_e262.Q OR _e263.Q) THEN Q_550M1 := TRUE; END_IF;
_e264(CLK := I_550Feed);
_e265(CLK := RebobinaAposNotOk);
IF P_On AND (_e264.Q OR _e265.Q) THEN Q_550M1 := FALSE; END_IF;

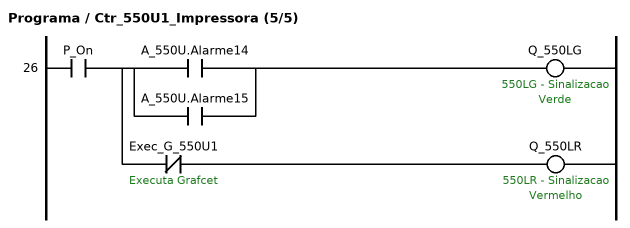
(* Rung 26 *)
Q_550LG := P_On AND (A_550U.Alarme14 OR A_550U.Alarme15);
Q_550LR := P_On AND NOT Exec_G_550U1;

(* Section Ctr_610M1: ladder, written here as Structured Text *)

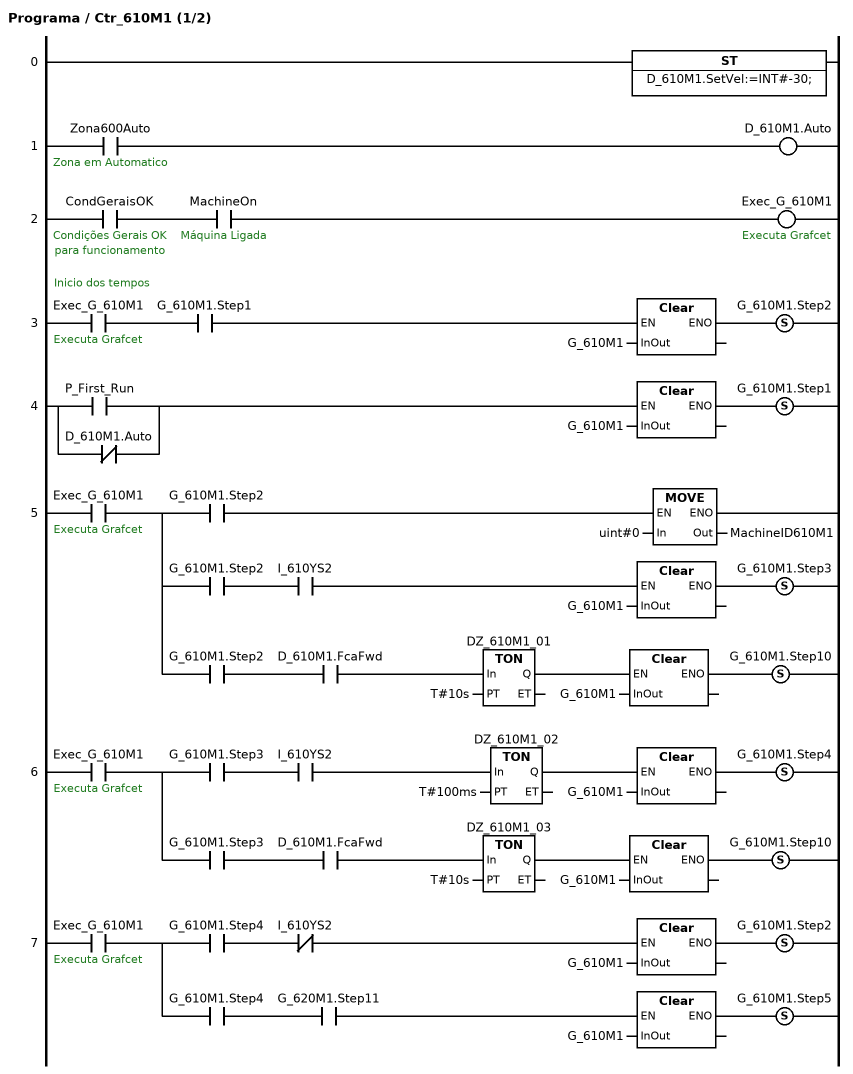
(* Rung 0 *)
D_610M1.SetVel:=INT#-30;
(* Rung 1 *)
D_610M1.Auto := Zona600Auto;
(* Rung 2 *)
Exec_G_610M1 := CondGeraisOK AND MachineOn;
(* Rung 3: Inicio dos tempos *)
_p266 := Exec_G_610M1 AND G_610M1.Step1;
IF _p266 THEN
    Clear(InOut := G_610M1);
    G_610M1.Step2 := TRUE;
END_IF;
(* Rung 4 *)
IF P_First_Run OR NOT D_610M1.Auto THEN
    Clear(InOut := G_610M1);
    G_610M1.Step1 := TRUE;
END_IF;
(* Rung 5 *)
IF Exec_G_610M1 AND G_610M1.Step2 THEN MachineID610M1 := uint#0; END_IF;
_p267 := Exec_G_610M1 AND G_610M1.Step2 AND I_610YS2;
IF _p267 THEN
    Clear(InOut := G_610M1);
    G_610M1.Step3 := TRUE;
END_IF;
DZ_610M1_01(In := Exec_G_610M1 AND G_610M1.Step2 AND D_610M1.FcaFwd, PT := T#10s);
IF DZ_610M1_01.Q THEN
    Clear(InOut := G_610M1);
    G_610M1.Step10 := TRUE;
END_IF;
(* Rung 6 *)
DZ_610M1_02(In := Exec_G_610M1 AND G_610M1.Step3 AND I_610YS2, PT := T#100ms);
IF DZ_610M1_02.Q THEN
    Clear(InOut := G_610M1);
    G_610M1.Step4 := TRUE;
END_IF;
DZ_610M1_03(In := Exec_G_610M1 AND G_610M1.Step3 AND D_610M1.FcaFwd, PT := T#10s);
IF DZ_610M1_03.Q THEN
    Clear(InOut := G_610M1);
    G_610M1.Step10 := TRUE;
END_IF;
(* Rung 7 *)
_p268 := Exec_G_610M1 AND G_610M1.Step4 AND NOT I_610YS2;
IF _p268 THEN
    Clear(InOut := G_610M1);
    G_610M1.Step2 := TRUE;
END_IF;
_p269 := Exec_G_610M1 AND G_610M1.Step4 AND G_620M1.Step11;
IF _p269 THEN
    Clear(InOut := G_610M1);
    G_610M1.Step5 := TRUE;
END_IF;

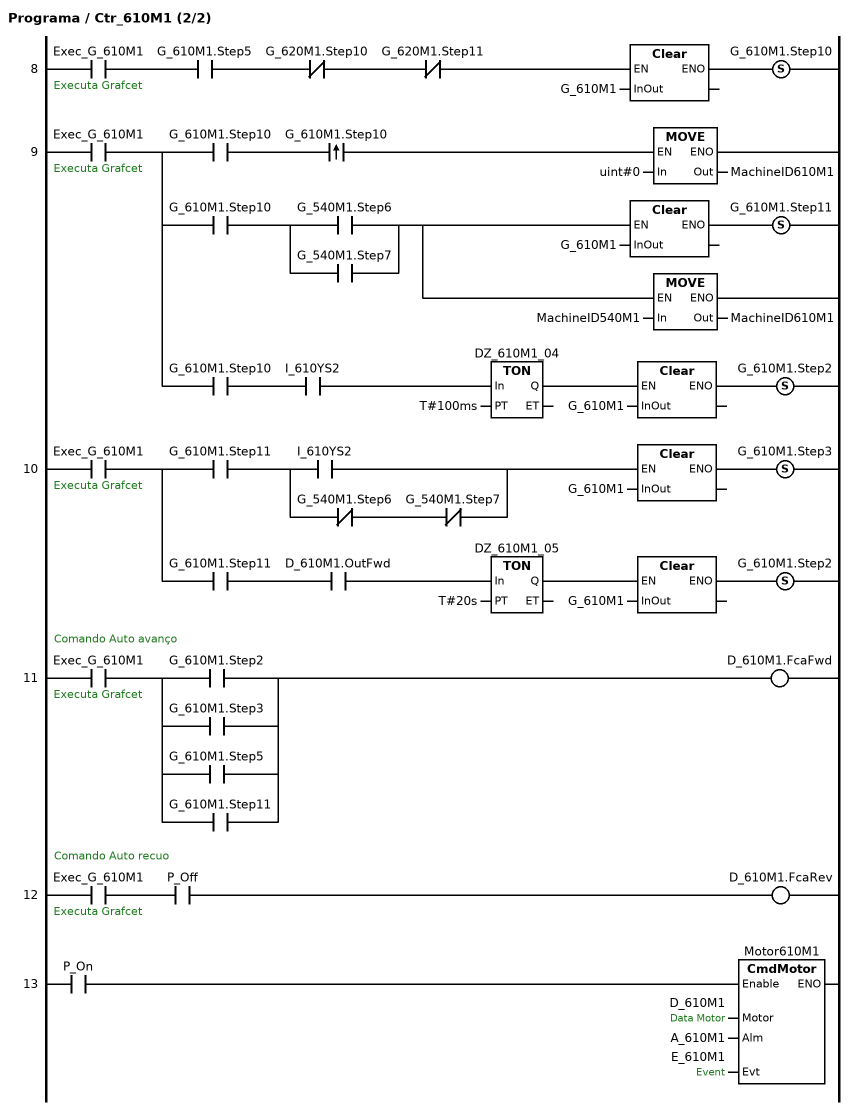
(* Rung 8 *)
_p270 := Exec_G_610M1 AND G_610M1.Step5 AND NOT G_620M1.Step10 AND NOT G_620M1.Step11;
IF _p270 THEN
    Clear(InOut := G_610M1);
    G_610M1.Step10 := TRUE;
END_IF;
(* Rung 9 *)
_e271(CLK := G_610M1.Step10);
IF Exec_G_610M1 AND G_610M1.Step10 AND _e271.Q THEN MachineID610M1 := uint#0; END_IF;
_p272 := Exec_G_610M1 AND G_610M1.Step10 AND (G_540M1.Step6 OR G_540M1.Step7);
IF _p272 THEN
    Clear(InOut := G_610M1);
    G_610M1.Step11 := TRUE;
    MachineID610M1 := MachineID540M1;
END_IF;
DZ_610M1_04(In := Exec_G_610M1 AND G_610M1.Step10 AND I_610YS2, PT := T#100ms);
IF DZ_610M1_04.Q THEN
    Clear(InOut := G_610M1);
    G_610M1.Step2 := TRUE;
END_IF;
(* Rung 10 *)
_p273 := Exec_G_610M1 AND G_610M1.Step11 AND (I_610YS2 OR (NOT G_540M1.Step6 AND NOT G_540M1.Step7));
IF _p273 THEN
    Clear(InOut := G_610M1);
    G_610M1.Step3 := TRUE;
END_IF;
DZ_610M1_05(In := Exec_G_610M1 AND G_610M1.Step11 AND D_610M1.OutFwd, PT := T#20s);
IF DZ_610M1_05.Q THEN
    Clear(InOut := G_610M1);
    G_610M1.Step2 := TRUE;
END_IF;
(* Rung 11: Comando Auto avanço *)
D_610M1.FcaFwd := Exec_G_610M1 AND (G_610M1.Step2 OR G_610M1.Step3 OR G_610M1.Step5 OR G_610M1.Step11);
(* Rung 12: Comando Auto recuo *)
D_610M1.FcaRev := Exec_G_610M1 AND P_Off;
(* Rung 13 *)
Motor610M1(Enable := P_On, Motor := D_610M1, Alm := A_610M1, Evt := E_610M1);

(* Section Ctr_620M1: ladder, written here as Structured Text *)

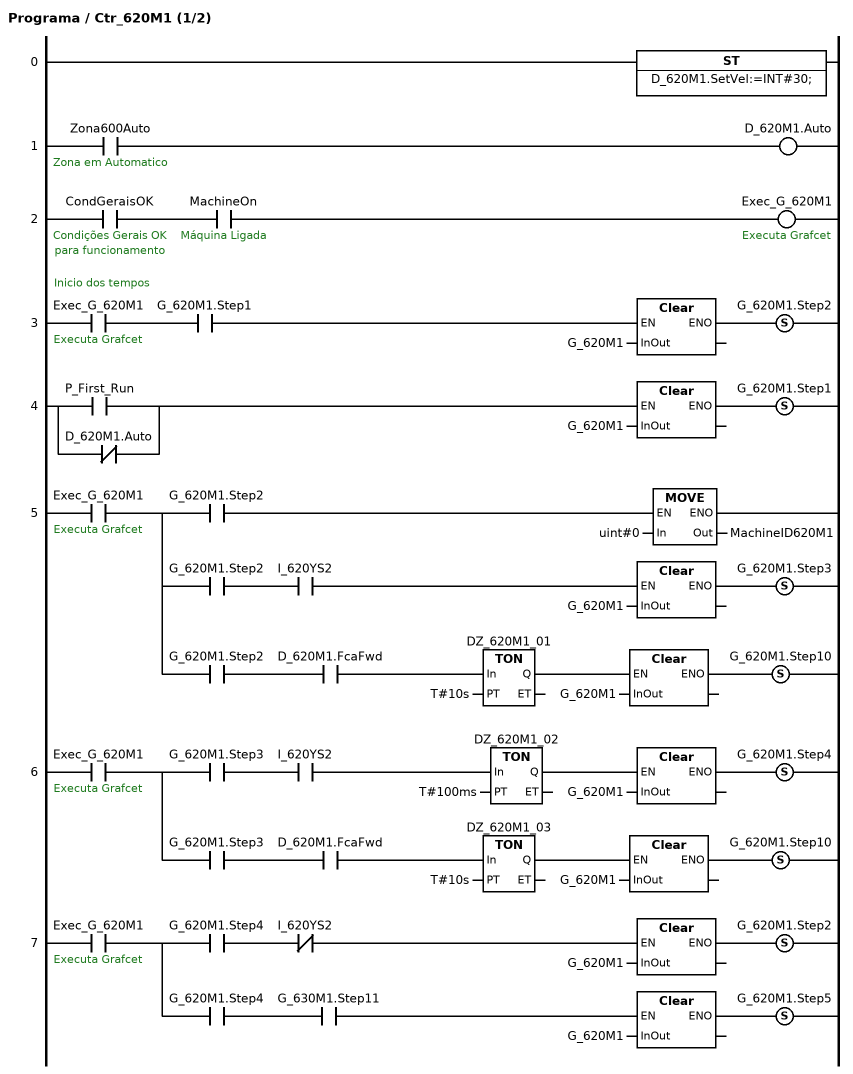
(* Rung 0 *)
D_620M1.SetVel:=INT#30;
(* Rung 1 *)
D_620M1.Auto := Zona600Auto;
(* Rung 2 *)
Exec_G_620M1 := CondGeraisOK AND MachineOn;
(* Rung 3: Inicio dos tempos *)
_p274 := Exec_G_620M1 AND G_620M1.Step1;
IF _p274 THEN
    Clear(InOut := G_620M1);
    G_620M1.Step2 := TRUE;
END_IF;
(* Rung 4 *)
IF P_First_Run OR NOT D_620M1.Auto THEN
    Clear(InOut := G_620M1);
    G_620M1.Step1 := TRUE;
END_IF;
(* Rung 5 *)
IF Exec_G_620M1 AND G_620M1.Step2 THEN MachineID620M1 := uint#0; END_IF;
_p275 := Exec_G_620M1 AND G_620M1.Step2 AND I_620YS2;
IF _p275 THEN
    Clear(InOut := G_620M1);
    G_620M1.Step3 := TRUE;
END_IF;
DZ_620M1_01(In := Exec_G_620M1 AND G_620M1.Step2 AND D_620M1.FcaFwd, PT := T#10s);
IF DZ_620M1_01.Q THEN
    Clear(InOut := G_620M1);
    G_620M1.Step10 := TRUE;
END_IF;
(* Rung 6 *)
DZ_620M1_02(In := Exec_G_620M1 AND G_620M1.Step3 AND I_620YS2, PT := T#100ms);
IF DZ_620M1_02.Q THEN
    Clear(InOut := G_620M1);
    G_620M1.Step4 := TRUE;
END_IF;
DZ_620M1_03(In := Exec_G_620M1 AND G_620M1.Step3 AND D_620M1.FcaFwd, PT := T#10s);
IF DZ_620M1_03.Q THEN
    Clear(InOut := G_620M1);
    G_620M1.Step10 := TRUE;
END_IF;
(* Rung 7 *)
_p276 := Exec_G_620M1 AND G_620M1.Step4 AND NOT I_620YS2;
IF _p276 THEN
    Clear(InOut := G_620M1);
    G_620M1.Step2 := TRUE;
END_IF;
_p277 := Exec_G_620M1 AND G_620M1.Step4 AND G_630M1.Step11;
IF _p277 THEN
    Clear(InOut := G_620M1);
    G_620M1.Step5 := TRUE;
END_IF;

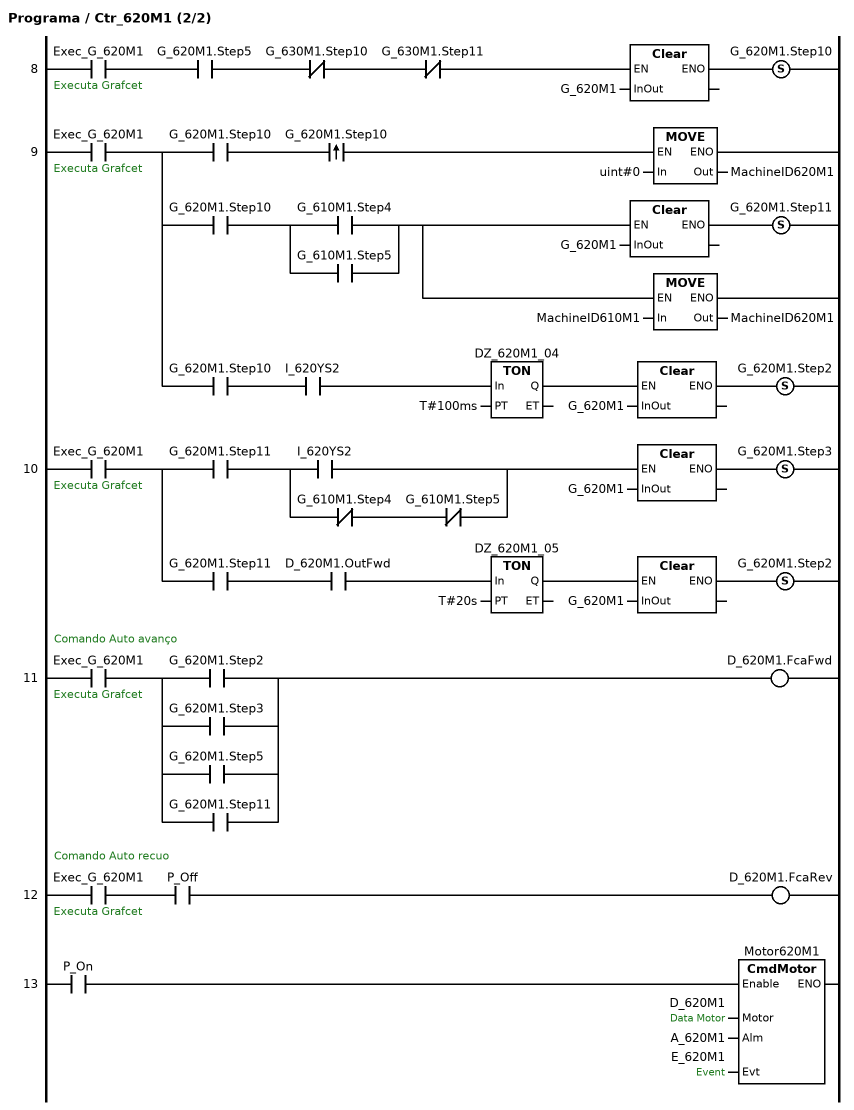
(* Rung 8 *)
_p278 := Exec_G_620M1 AND G_620M1.Step5 AND NOT G_630M1.Step10 AND NOT G_630M1.Step11;
IF _p278 THEN
    Clear(InOut := G_620M1);
    G_620M1.Step10 := TRUE;
END_IF;
(* Rung 9 *)
_e279(CLK := G_620M1.Step10);
IF Exec_G_620M1 AND G_620M1.Step10 AND _e279.Q THEN MachineID620M1 := uint#0; END_IF;
_p280 := Exec_G_620M1 AND G_620M1.Step10 AND (G_610M1.Step4 OR G_610M1.Step5);
IF _p280 THEN
    Clear(InOut := G_620M1);
    G_620M1.Step11 := TRUE;
    MachineID620M1 := MachineID610M1;
END_IF;
DZ_620M1_04(In := Exec_G_620M1 AND G_620M1.Step10 AND I_620YS2, PT := T#100ms);
IF DZ_620M1_04.Q THEN
    Clear(InOut := G_620M1);
    G_620M1.Step2 := TRUE;
END_IF;
(* Rung 10 *)
_p281 := Exec_G_620M1 AND G_620M1.Step11 AND (I_620YS2 OR (NOT G_610M1.Step4 AND NOT G_610M1.Step5));
IF _p281 THEN
    Clear(InOut := G_620M1);
    G_620M1.Step3 := TRUE;
END_IF;
DZ_620M1_05(In := Exec_G_620M1 AND G_620M1.Step11 AND D_620M1.OutFwd, PT := T#20s);
IF DZ_620M1_05.Q THEN
    Clear(InOut := G_620M1);
    G_620M1.Step2 := TRUE;
END_IF;
(* Rung 11: Comando Auto avanço *)
D_620M1.FcaFwd := Exec_G_620M1 AND (G_620M1.Step2 OR G_620M1.Step3 OR G_620M1.Step5 OR G_620M1.Step11);
(* Rung 12: Comando Auto recuo *)
D_620M1.FcaRev := Exec_G_620M1 AND P_Off;
(* Rung 13 *)
Motor620M1(Enable := P_On, Motor := D_620M1, Alm := A_620M1, Evt := E_620M1);

(* Section Ctr_630M1: ladder, written here as Structured Text *)

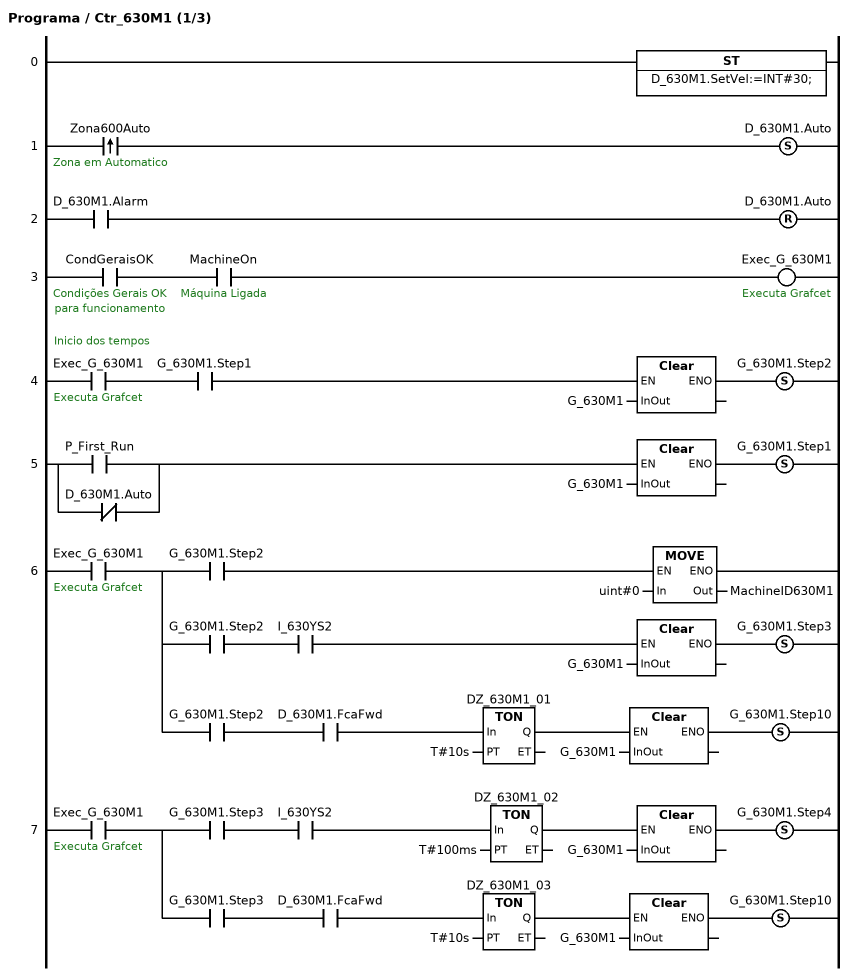
(* Rung 0 *)
D_630M1.SetVel:=INT#30;
(* Rung 1 *)
_e282(CLK := Zona600Auto);
IF _e282.Q THEN D_630M1.Auto := TRUE; END_IF;
(* Rung 2 *)
IF D_630M1.Alarm THEN D_630M1.Auto := FALSE; END_IF;
(* Rung 3 *)
Exec_G_630M1 := CondGeraisOK AND MachineOn;
(* Rung 4: Inicio dos tempos *)
_p283 := Exec_G_630M1 AND G_630M1.Step1;
IF _p283 THEN
    Clear(InOut := G_630M1);
    G_630M1.Step2 := TRUE;
END_IF;
(* Rung 5 *)
IF P_First_Run OR NOT D_630M1.Auto THEN
    Clear(InOut := G_630M1);
    G_630M1.Step1 := TRUE;
END_IF;
(* Rung 6 *)
IF Exec_G_630M1 AND G_630M1.Step2 THEN MachineID630M1 := uint#0; END_IF;
_p284 := Exec_G_630M1 AND G_630M1.Step2 AND I_630YS2;
IF _p284 THEN
    Clear(InOut := G_630M1);
    G_630M1.Step3 := TRUE;
END_IF;
DZ_630M1_01(In := Exec_G_630M1 AND G_630M1.Step2 AND D_630M1.FcaFwd, PT := T#10s);
IF DZ_630M1_01.Q THEN
    Clear(InOut := G_630M1);
    G_630M1.Step10 := TRUE;
END_IF;
(* Rung 7 *)
DZ_630M1_02(In := Exec_G_630M1 AND G_630M1.Step3 AND I_630YS2, PT := T#100ms);
IF DZ_630M1_02.Q THEN
    Clear(InOut := G_630M1);
    G_630M1.Step4 := TRUE;
END_IF;
DZ_630M1_03(In := Exec_G_630M1 AND G_630M1.Step3 AND D_630M1.FcaFwd, PT := T#10s);
IF DZ_630M1_03.Q THEN
    Clear(InOut := G_630M1);
    G_630M1.Step10 := TRUE;
END_IF;

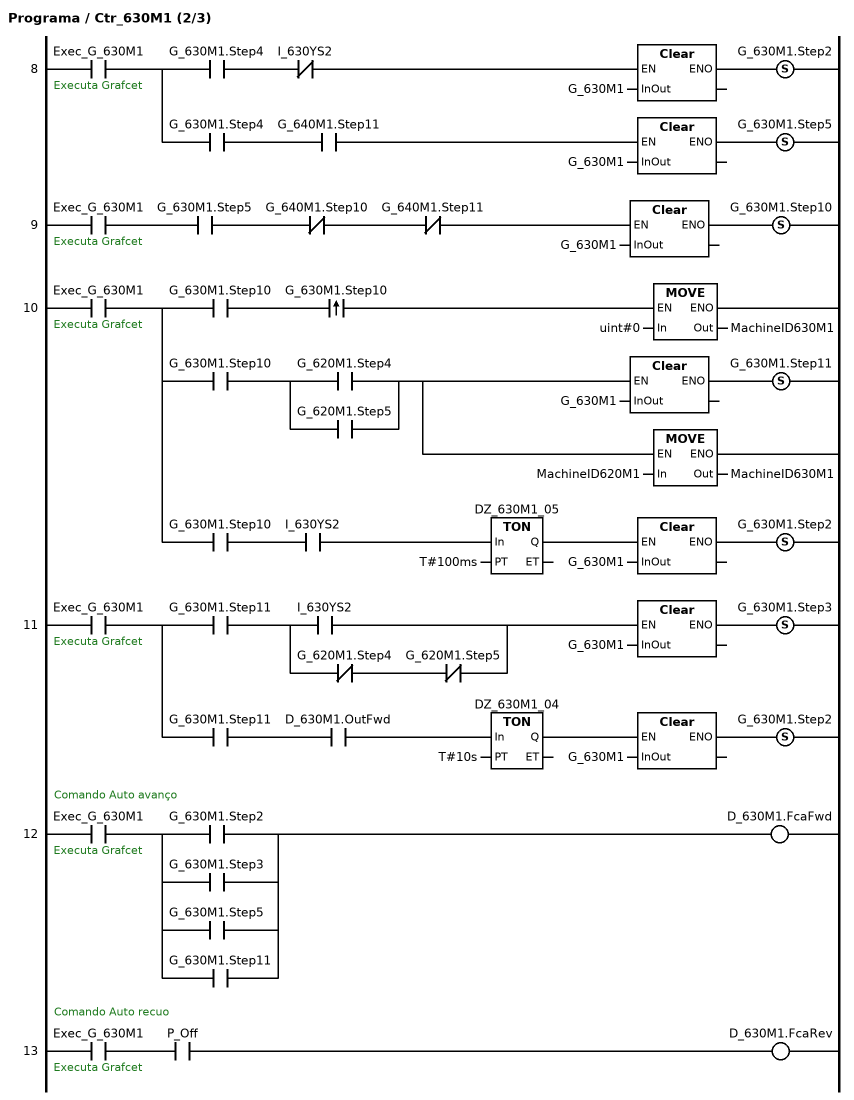
(* Rung 8 *)
_p285 := Exec_G_630M1 AND G_630M1.Step4 AND NOT I_630YS2;
IF _p285 THEN
    Clear(InOut := G_630M1);
    G_630M1.Step2 := TRUE;
END_IF;
_p286 := Exec_G_630M1 AND G_630M1.Step4 AND G_640M1.Step11;
IF _p286 THEN
    Clear(InOut := G_630M1);
    G_630M1.Step5 := TRUE;
END_IF;
(* Rung 9 *)
_p287 := Exec_G_630M1 AND G_630M1.Step5 AND NOT G_640M1.Step10 AND NOT G_640M1.Step11;
IF _p287 THEN
    Clear(InOut := G_630M1);
    G_630M1.Step10 := TRUE;
END_IF;
(* Rung 10 *)
_e288(CLK := G_630M1.Step10);
IF Exec_G_630M1 AND G_630M1.Step10 AND _e288.Q THEN MachineID630M1 := uint#0; END_IF;
_p289 := Exec_G_630M1 AND G_630M1.Step10 AND (G_620M1.Step4 OR G_620M1.Step5);
IF _p289 THEN
    Clear(InOut := G_630M1);
    G_630M1.Step11 := TRUE;
    MachineID630M1 := MachineID620M1;
END_IF;
DZ_630M1_05(In := Exec_G_630M1 AND G_630M1.Step10 AND I_630YS2, PT := T#100ms);
IF DZ_630M1_05.Q THEN
    Clear(InOut := G_630M1);
    G_630M1.Step2 := TRUE;
END_IF;
(* Rung 11 *)
_p290 := Exec_G_630M1 AND G_630M1.Step11 AND (I_630YS2 OR (NOT G_620M1.Step4 AND NOT G_620M1.Step5));
IF _p290 THEN
    Clear(InOut := G_630M1);
    G_630M1.Step3 := TRUE;
END_IF;
DZ_630M1_04(In := Exec_G_630M1 AND G_630M1.Step11 AND D_630M1.OutFwd, PT := T#10s);
IF DZ_630M1_04.Q THEN
    Clear(InOut := G_630M1);
    G_630M1.Step2 := TRUE;
END_IF;
(* Rung 12: Comando Auto avanço *)
D_630M1.FcaFwd := Exec_G_630M1 AND (G_630M1.Step2 OR G_630M1.Step3 OR G_630M1.Step5 OR G_630M1.Step11);
(* Rung 13: Comando Auto recuo *)
D_630M1.FcaRev := Exec_G_630M1 AND P_Off;

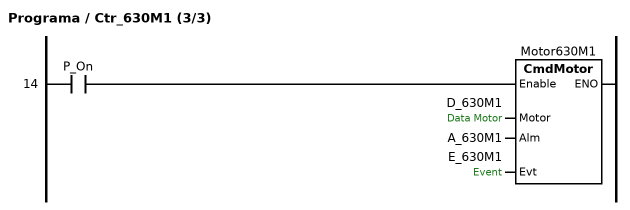
(* Rung 14 *)
Motor630M1(Enable := P_On, Motor := D_630M1, Alm := A_630M1, Evt := E_630M1);

(* Section Ctr_640M1: ladder, written here as Structured Text *)

